FUNCTION_BLOCK "GCS7_E_AnalogInput"	// FB 19
TITLE = Analog Input
//  
//COPYRIGHT:    (C) 2000 BY  BUHLER AG,  CH-9240 UZWILn  SWITZERLAND
//
//PRODUCT:      GCS7
//
//TITLE:        Element Analog Input
//
//-------------------------------------------------------------------------
//
//IDENT:        AUTHOR:             DEPT:                       DATE:
//
//FB19.1.5      A. Egli             CT3                         06-Oct-2008
//              ParMonTimeL=0 or ParMonTimeH=0 are also valide values
//FB19.1.4      A. Egli             CT3                         08-Mar-2005
//              Check ParLimitL > ParLimitLL and ParLimitH < ParLimitHH
//FB19.1.3      A. Egli             CT3                         24-Jan-2005
//              InDisable
//FB19.1.2      A. Egli             CT3                         26-Nov-2001
//              PCDirect Control: Length data is 80 byte not 40 
//FB19.1.1      A. Egli             CT3                         26-Nov-2001
//              Transition StL -->StLL ,StH -->StHH
//FB19.1.0      A. Egli             CT3                         22-Oct-2001
//              New Version of Anlaog Input
//
//-------------------------------------------------------------------------
//
//PURPOSE:      MANUAL : see [AIxxMAN]
//
//RESTRICTIONS: Use the CALL command to call the element
//              e.g. CALL "Element1"
//
//-------------------------------------------------------------------------
//
//MaxDigits:     Siemens: 27'648/ Wago: 32'767
//
//=======================================================
//Log Message: 
//------------------------------------------------------
//1StLLrange LL
//2StLrange L
//3StMidrange Mid
//4StHrange H
//5StHHrange HH
//7fault AI
//8fault device
//9fault cancelled
//11prealarm LL
//12prealarm LL
//13prealarm LL
//14prealarm LL
//15prealarm HH
//21fault LL
//22fault L
//23fault Mid
//24fault H
//25fault HH
//
//=======================================================
//StCode:  State               
//------------------------------------------------------
//  1   StLL                      range LL
//  2   StL                       range L
//  3   StMiddle                  range middle
//  4   StH                       range H
//  5   StHH                      range HH
//
// 11   StLL.Warning              range LL Warning
// 12   StL.Warning               range L  Warning 
// 13   StMiddle                  range middle Warning
// 14   StH.Warning               range H  Warning
// 15   StHH.Warning              range HH Warning
//
// 21   StLL.Faulted              range LL Faulted
// 22   StL.Faulted               range L  Faulted
// 23   StMiddle.Faulted          range middle Faulted
// 24   StH.Faulted               range H  Faulted 
// 25   StHH.Faulted              range HH Faulted
//
// 41   StLL.HWStop               range LL HWStop
// 42   StL.HWStop                range L  HWStop
// 43   StMiddle.HWStop           range middle HWStop
// 44   StH..HWStop               range H  HWStop
// 45   StHH..HWStop              range HH HWStop
//
// 51   StLL.DPFault              range LL DPFault
// 52   StL.DPFault               range L  DPFault
// 53   StMiddle.DPFault          range middle DPFault
// 54   StH..DPFault              range H  DPFault
// 55   StHH..DPFault             range HH DPFault
//
//
// 29   StFaultAI.Dev             fault Device Passiv
// 30   StFaultAI.Input           fault Input  Passiv
// 31   StFaultAI.Dev             fault Device Active
// 32   StFaultAI.Input           fault Input  Active
//
//
//
AUTHOR : EA
FAMILY : GCS7LL
NAME : EL_AI2
VERSION : 1.5
VAR
  StCode : INT ;	//Element state code
  InMonLL : BOOL ;	//After t1 value must be <>StLL, otherwise it is a process fault
  InMonL : BOOL ;	//After t2 value must be <>StL, otherwise it is a process fault
  InMonMid : BOOL ;	//After t3 value must be <>StMid, otherwise it is a process fault
  InMonH : BOOL ;	//After t4 value must be <>StH, otherwise it is a process fault
  InMonHH : BOOL ;	//After t5 value must be <>StHH, otherwise it is a process fault
  spare0205 : BOOL ;
  InpFaultAI : BOOL ;	//Digital input:Fault A/D converter WAGO
  InpFaultDev : BOOL ;	//Digital input Fault device
  InHWStop : BOOL ;	//HW stop is detected, no fault
  InDPFault : BOOL ;	//DP-Fault is detected, no fault
  InDisable : BOOL ;	//Element is disabled
  CmdFaultReset : BOOL ;	//Command to reset fault
  InLocal : BOOL ;	//Local mode
  spare0305 : BOOL ;
  InReport : BOOL ;	//Report all state transitions
  spare0307 : BOOL ;
  OutLL : BOOL ;	//Internal used InValue >= Limit Low Low
  OutL : BOOL ;	//Internal used InValue >= Limit Low
  OutH : BOOL ;	//Internal used InValue >= Limit High
  OutHH : BOOL ;	//Internal used InValue >= Limit High High
  OutOverflow : BOOL ;	//InpValue >32767
  spare0405 : BOOL ;
  OutFaultAI : BOOL ;	//Fault analog input signal
  spare0407 : BOOL ;
  StLL : BOOL ;	//InValue < ParLimitLL (with delay time)
  StL : BOOL ;	//InValue < ParLimitL  (with delay time)
  StMid : BOOL ;	//ParLimitL < InValue < ParLimitH (with delay time)
  StH : BOOL ;	//InValue  > ParLimitH (with delay time)
  StHH : BOOL ;	//InValue  > ParLimitHH (with delay time)
  StFaultAI : BOOL ;	//Fault of analog input value (InpFaultDev or OutFaultAI)
  OutWarning : BOOL ;	//Substate StCode Xxxx.Warning
  OutFaulted : BOOL ;	//Substate StCode Xxxx.Fault
  InpValue : INT ;	//Actual value of analog input
  OutValuePc : INT ;	//Converted InValue in [0.01 %]
  OutValueUnits : DINT ;	//Converted InValue in units
  Msg : STRUCT 	//Read by WinCC
   WarningDoneLL : BOOL ;
   WarningDoneL : BOOL ;
   WarningDoneMid : BOOL ;
   WarningDoneH : BOOL ;
   WarningDoneHH : BOOL ;
   FaultDoneLL : BOOL ;
   FaultDoneL : BOOL ;
   FaultDoneMid : BOOL ;
   FaultDoneH : BOOL ;
   FaultDoneHH : BOOL ;
   FaultDoneDev : BOOL ;
   FaultDoneAI : BOOL ;
  END_STRUCT ;
  OutAlarmNrLog : INT ;	//Last textnumber send to log
  Par : STRUCT
   ParObjectNo : INT ;	//Is used for communication with PC, e.g. for message
   ParMsgType : INT ;	//Is used for message (translation of state)
   ParHornCode : INT ;	//Is used by horn module
   ParLogOff : BOOL ;	//Report is off
   ParSpare0401 : BOOL ;
   ParValueByUser : BOOL ;	//User writes value direct to OutValueUnits
   ParLimitsPc : BOOL ;	//Limits in percent not in units.
   ParWago : BOOL ;	//Format of analog value is WAGO
   ParNoHornByWarning : BOOL ;	//No alarm horn by warning
   ParWarningLL : BOOL ;	//1=Warning / 0=Fault
   ParWarningL : BOOL ;	//1=Warning / 0=Fault
   ParWarningMid : BOOL ;	//1=Warning / 0=Fault
   ParWarningH : BOOL ;	//1=Warning / 0=Fault
   ParWarningHH : BOOL ;	//1=Warning / 0=Fault
   ParPreAlarmLL : BOOL ;	//Immediately Alarm (Horn and report), if value out of monitored range (after t0.
   ParPreAlarmL : BOOL ;	//Immediately Alarm (Horn and report), if value out of monitored range (after t0.
   ParPreAlarmMid : BOOL ;	//Immediately Alarm (Horn and report), if value out of monitored range (after t0.
   ParPreAlarmH : BOOL ;	//Immediately Alarm (Horn and report), if value out of monitored range (after t0.
   ParPreAlarmHH : BOOL ;	//Immediately Alarm (Horn and report), if value out of monitored range (after t0.
   ParUnitsByZeroDigit : DINT ;	//Zero set point of AD-Converter in units
   ParUnitsByMaxDigit : DINT ;	//Max set point of AD-Converter in units
   ParUnitsBy100Pc : DINT ;	//100 Pc set point of precess working range in units
   ParLimitLL : DINT ;	//LL limit value in units or percent
   ParLimitL : DINT ;	//L limit value in units or percent
   ParLimitH : DINT ;	//H limit value in units or percent
   ParLimitHH : DINT ;	//HH limit value in units or percent
   ParMonTimeLL : INT ;	//t1: At end of t1 InValue has to be <> StLL, otherwise StFault.
   ParMonTimeL : INT ;	//t1: At end of t1 InValue has to be <> StL, otherwise StFault.
   ParMonTimeMid : INT ;	//t2: At end of t2 InValue has to be <> StMid, otherwise StFault.
   ParMonTimeH : INT ;	//t2: At end of t2 InValue has to be <> StH, otherwise StFault.
   ParMonTimeHH : INT ;	//t3: At end of t3 InValue has to be <> StHH, otherwise StFault.
   ParDelayTimeDown : INT  := 20;	//Delay time until element changes to the lower state
   ParDelayTimeUp : INT  := 20;	//Delay time until element changes to the higher state
   ParDelayTime : INT ;	//Requested fault delay time (InpFaultAI, InpFaultDev)
   OutMonTimeLL : INT ;	//Actual time: monitoring
   OutMonTimeL : INT ;	//Actual time: monitoring
   OutMonTimeMid : INT ;	//Actual time: monitoring
   OutMonTimeH : INT ;	//Actual time: monitoring
   OutMonTimeHH : INT ;	//Actual time: monitoring
   OutDelayTimeDown : INT ;	//Actual time: delay
   OutDelayTimeUp : INT ;	//Actual time: delay
   OutDelayTime : INT ;	//Actual time: DelayTime
   Spare66 : INT ;
  END_STRUCT ;
END_VAR
VAR_TEMP
  tmpStoreAR2 : DWORD ;	//store the Instance Pointer
  tmpLenDyn : DINT ;
  tmpLOGvalue : WORD ;	//LOG value
  tmpReport : BOOL ;	//Global LOG all
  tmpDConverter : REAL ;	//provisional result: ParUnitsByMaxDigit - ParUnitsByZeroDigit
  tmpDProcess : REAL ;	//provisional result: ParUnitsBy100Pc - ParUnitsByZeroDigit
  tmpLimitMinPc : REAL ;	//Limit minimum in percent
  tmpLimitMaxPc : REAL ;	//Limit maximum in percent
  tmpInpValue : REAL ;	//store actual value
  tmpFaultAI : BOOL ;
  tmpLocal : BOOL ;
  tmpHornOn : BOOL ;
END_VAR
BEGIN
NETWORK
TITLE = Start Global
      L     88;
      T     #tmpLenDyn;	//--> Len dynamic data in byte
//---Report is on---
      O     "GCS7_Gr_OutReportAll";	//---Global OutReportAll
      O     #InReport;
      =     #tmpReport;
//--Local ------------
      A     #InLocal;
      O     #InHWStop;
      O     #InDPFault;
      O     #InDisable;	//[1.3]
      =     #tmpLocal;
//-----------------
      SET;
      R     #tmpHornOn;
NETWORK
TITLE = PC Control
      L     "SYS_DirectCtrlDB".PC.ObjectNo;	//PCControl.ObjectNo
      L     #Par.ParObjectNo;	//Input ObjectNo
      <>I;
      JC    Ctrl;
//=== Test OType      ========================
      L     1019;	//Input object type
      L     "SYS_DirectCtrlDB".PC.ObjectType;	//PCControl.ObjectType
      <>I;
      JC    Ctrl;
//=== Test Handshake =========================
      A     "SYS_DirectCtrlDB".PC.Hsk.FExamine;	//PC.Hsk.FExamine
      JC    pExa;
      A     "SYS_DirectCtrlDB".PC.Hsk.FDefineCmd;	// PC.Hsk.FDefineCmd
      JC    pCmd;
      A     "SYS_DirectCtrlDB".PC.Hsk.FDefinePara;	//PC.Hsk.FDefinePara
      JC    pPar;
pIni: L     2;	// FcInit
      UC    "SYS_DirectCtrl";
      JU    Ctrl;
// Write parameter 
pPar: LAR1  P#DBX 58.0;
      L     P##Par;
      L     DW#16#FFFFF;
      AD;
      +AR1;
      L     DBD [AR1,P#20.0];
      T     #Par.ParLimitLL;
      L     DBD [AR1,P#24.0];
      T     #Par.ParLimitL;
      L     DBD [AR1,P#28.0];
      T     #Par.ParLimitH;
      L     DBD [AR1,P#32.0];
      T     #Par.ParLimitHH;
      L     DBW [AR1,P#36.0];
      T     #Par.ParMonTimeLL;
      L     DBW [AR1,P#38.0];
      T     #Par.ParMonTimeL;
      L     DBW [AR1,P#40.0];
      T     #Par.ParMonTimeMid;
      L     DBW [AR1,P#42.0];
      T     #Par.ParMonTimeH;
      L     DBW [AR1,P#44.0];
      T     #Par.ParMonTimeHH;
      L     DBW [AR1,P#46.0];
      T     #Par.ParDelayTimeDown;
      L     DBW [AR1,P#48.0];
      T     #Par.ParDelayTimeUp;
      L     DBW [AR1,P#50.0];
      T     #Par.ParDelayTime;
// Write new commands from PC to Interface object
pCmd: A     "SYS_DirectCtrlDB".PC.Cmd1[11];	//Cmd1[11]=CmdFaultReset
      S     #CmdFaultReset;
      A     "SYS_DirectCtrlDB".PC.Cmd1[14];	//Cmd1[14]=CmdReportOn
      S     #InReport;
      A     "SYS_DirectCtrlDB".PC.Cmd2[14];	//Cmd2[14]=CmdReportOff
      R     #InReport;
      JU    pIni;
pExa: TAR2;	// Address Dynamic datas
      T     "SYS_DirectCtrlDB".GC.InDynAddr;	// -->PCControl.GC.InDynAddr
      L     #tmpLenDyn;	// Length Dynamic datas
      T     "SYS_DirectCtrlDB".GC.InDynLen;	// -->PCControl.GC.InDynLen
      L     "SYS_DirectCtrlDB".GC.InDynAddr;	// Address Parameters
      T     "SYS_DirectCtrlDB".GC.InParaAddr;	// -->PCControl.GC.InParaAddr
      L     0;	// Length parameter
      T     "SYS_DirectCtrlDB".GC.InParaLen;	// -->PCControl.GC.InParaLen
      L     1;	// Code FcExamine
      UC    "SYS_DirectCtrl";
Ctrl: NOP   0;
NETWORK
TITLE = Global Value Calculation
//                   InpValue    
// OutValueUnits =   -------- * (ParUnitsByMaxDigit- ParUnitsByZeroDigit) 
//+ParUnitsByZeroDigit
//                   maxDigits     
//                     
// OutValuePc    =   (OutValueUnits / ParUnitsBy100Pc) *10'000
//                     
      AN    #Par.ParValueByUser;
      JC    aiJ1;
      L     #OutValueUnits;	// Value by user software
      DTR;
      JU    aiPc;
aiJ1: L     32767;
      L     #InpValue;
      ==I;
      AN    #Par.ParWago;
      =     #OutOverflow;
      L     -32767;
      <=I;
      AN    #Par.ParWago;
      O     #InpFaultAI;
      =     #OutFaultAI;	//--> Wireing broken of underflow analog input
      L     0.000000e+00;
      JC    aiNO;	// aip0
      L     #InpValue;
      ITD;
      DTR;
      A     #Par.ParWago;
      JC    aiJw;
      L     2.764800e+04;	// Max number of digits SIEMENS          
      JU    aiJc;
aiJw: L     3.276700e+04;	// Max number of digits WAGO             
aiJc: /R;
      T     #tmpInpValue;
      L     #Par.ParUnitsByMaxDigit;
      L     #Par.ParUnitsByZeroDigit;
      -D;
      DTR;
      L     #tmpInpValue;
      *R;
      L     #Par.ParUnitsByZeroDigit;
      DTR;
      +R;
      T     #tmpInpValue;
      RND;	// Real to Integer
      T     #OutValueUnits;
      L     #tmpInpValue;
aiPc: L     #Par.ParUnitsBy100Pc;
      DTR;
      /R;
      L     1.000000e+04;
      *R;
      RND;	// Real to Integer
      T     #OutValuePc;
aiNO: NOP   0;
NETWORK
TITLE = Test limits
      L     #OutValuePc;
      ITD;
      A     #Par.ParLimitsPc;
      JC    bLL;
      L     #OutValueUnits;
bLL:  L     #Par.ParLimitLL;
      >=D;
      =     #OutLL;
// 
      L     #OutValuePc;
      ITD;
      A     #Par.ParLimitsPc;
      JC    bL;
      L     #OutValueUnits;
bL:   L     #Par.ParLimitL;
      >=D;
      A     #OutLL;	//[1.4]
      =     #OutL;
// 
      L     #OutValuePc;
      ITD;
      A     #Par.ParLimitsPc;
      JC    bHH;
      L     #OutValueUnits;
bHH:  L     #Par.ParLimitHH;
      >D;
      =     #OutHH;
// 
      L     #OutValuePc;
      ITD;
      A     #Par.ParLimitsPc;
      JC    bH;
      L     #OutValueUnits;
bH:   L     #Par.ParLimitH;
      >D;
      O     #OutHH;	//[1.4]
      =     #OutH;
//---Report is on---
      O     "GCS7_Gr_OutReportAll";	//---Global OutReportAll
      O     #InReport;
      =     #tmpReport;
NETWORK
TITLE = Fault delay time: ParDelayTime 
//Test or Running delay time ====================
//---Condition for Delay Fault
      A     #InpFaultDev;
      O     #OutFaultAI;
      AN    #tmpLocal;
      JC    TFF1;
      R     #tmpFaultAI;
      L     0;
      T     #Par.OutDelayTime;
      JU    TFF0;
TFF1: AN    "GCS7_Gr_OutTick200ms";	// Decrement all 200ms
      L     #Par.OutDelayTime;
      JC    TFF3;
      +     2;
TFF3: T     #Par.OutDelayTime;
      L     #Par.ParDelayTime;
      >=I;
      =     #tmpFaultAI;
      JCN   TFF0;
      T     #Par.OutDelayTime;
TFF0: NOP   0;
NETWORK
TITLE = Count Delay Timer
      AN    "GCS7_Gr_OutTick500ms";	//Gr.OutTick500ms
      JC    DTJ0;
      L     #Par.OutDelayTimeDown;
      +     5;	//Increment all 500ms
      T     #Par.OutDelayTimeDown;
      L     #Par.OutDelayTimeUp;
      +     5;	//Increment all 500ms
      T     #Par.OutDelayTimeUp;
DTJ0: NOP   0;
NETWORK
TITLE = FaultReset
      AN    #CmdFaultReset;	//---Condition for StFault
      AN    "GCS7_Gr_OutFaultReset";	// Gr.OutFaultReset
      AN    #InLocal;
      JC    FREn;
      R     #Msg.WarningDoneLL;
      R     #Msg.WarningDoneL;
      R     #Msg.WarningDoneMid;
      R     #Msg.WarningDoneH;
      R     #Msg.WarningDoneHH;
      R     #Msg.FaultDoneLL;
      R     #Msg.FaultDoneL;
      R     #Msg.FaultDoneMid;
      R     #Msg.FaultDoneH;
      R     #Msg.FaultDoneHH;
      R     #Msg.FaultDoneAI;
      R     #Msg.FaultDoneDev;
//--- Message Fault Cancelled---------------
      A     #Par.ParLogOff;
      ON    #OutFaulted;
      R     #OutFaulted;
      JC    FREn;
      R     #OutFaulted;
      L     B#(3, 9);	// MessageClass Operater "fault cancelled"
      T     #tmpLOGvalue;
      CALL  "GCS7_LogConvert" (
           ObjectNo                 := #Par.ParObjectNo,
           MsgType                  := #Par.ParMsgType,
           ClassMsgTxt              := #tmpLOGvalue,
           OType                    := 1019);	// LOG Message Converter / Entry / Contains Class and TextNo
FREn: NOP   0;
NETWORK
TITLE = Init States
      AN    #StLL;
      AN    #StL;
      AN    #StMid;
      AN    #StH;
      AN    #StHH;
      AN    #StFaultAI;
      JCN   InEn;
///=====================================
//Init after download DB
///=====================================
//Condition for StHH
      A     #OutHH;
      JC    xxHH;
//Condition for StH
      A     #OutH;
      JC    xx_H;
//Condition for StMid
      A     #OutL;
      JC    xxMi;
//Condition for StL
      A     #OutLL;
      JC    xx_L;
//Condition for StLL
      JU    xxLL;
InEn: NOP   0;
NETWORK
TITLE = StLL
      AN    #StLL;
      JC    LLEn;
      JU    LL;
//===============================================
//Transition  to StLL
//===============================================
xxLL: SET;
      S     #StLL;	//Initialise: goto StLL
      L     0;
      T     #Par.OutDelayTimeUp;
      AN    #InReport;
      JC    LLEn;
      L     B#(4, 1);	// Message ('Low Low' )
      JU    Log;
//===============================================
//Logic
//===============================================
//Init
LL:   AN    #InMonLL;
      R     #OutWarning;
      L     0;
      T     #Par.OutDelayTimeDown;
      A     #OutLL;
      JC    LLJ1;
      L     0;
      T     #Par.OutDelayTimeUp;
//---1. Condition for StFault
LLJ1: A     #tmpFaultAI;
      R     #StLL;
      JC    xxFI;
//---Condition for StL
      L     #Par.ParDelayTimeUp;
      L     #Par.OutDelayTimeUp;
      <=I;
      A     #OutLL;	//Change with delay
      O     #OutL;	//Immediate change
      R     #StLL;
      JC    xx_L;
LLEn: NOP   0;
NETWORK
TITLE = Monitoring LL
      AN    #OutLL;
      A     #InMonLL;
      AN    #tmpLocal;
      JC    mLL1;
      L     #Par.ParMonTimeLL;
      T     #Par.OutMonTimeLL;
      JU    mLL0;
mLL1: AN    "GCS7_Gr_OutTick500ms";	//Gr.OutTick500ms
      L     #Par.OutMonTimeLL;
      JC    mLL2;
      L     5;
      -I;	// Decrement all 500ms
      JP    mLL2;
      L     0;
mLL2: T     #Par.OutMonTimeLL;
//----------------------------------------
//FaultLL
//----------------------------------------
      L     #Par.OutMonTimeLL;
      L     0;
      <=I;
      AN    #Par.ParWarningLL;
      JCN   mLLP;
      S     #OutFaulted;
      AN    #Msg.FaultDoneLL;
      S     #Msg.FaultDoneLL;
      S     #tmpHornOn;
      L     B#(1, 21);	// MessageClass Error "fault Low Low"
      JC    Log;
//----------------------------------------
//PreAlarm/WarningLL
//----------------------------------------
mLLP: L     #Par.OutMonTimeLL;
      L     0;
      <=I;
      O     #Par.ParPreAlarmLL;
      JCN   mLL0;
      S     #OutWarning;
      AN    #Msg.FaultDoneLL;
      AN    #Msg.WarningDoneLL;
      JCN   mLL0;
      S     #Msg.WarningDoneLL;
      AN    #Par.ParNoHornByWarning;
      S     #tmpHornOn;
      L     B#(1, 11);	// MessageClass Error "warning Low Low"
      JC    Log;
mLL0: NOP   0;
NETWORK
TITLE = StL
      AN    #StL;
      JC    _LEn;
      JU    _L;
//===============================================
//Transition  to StL
//===============================================
xx_L: SET;
      S     #StL;
      R     #Msg.WarningDoneLL;
      L     0;
      T     #Par.OutDelayTimeDown;
      T     #Par.OutDelayTimeUp;
      AN    #InReport;
      JC    _LEn;
      L     B#(4, 2);	// Message ('Low' )
      JU    Log;
//===============================================
//Logic
//===============================================
//Init
_L:   AN    #InMonL;
      R     #OutWarning;
      AN    #OutLL;
      JC    _LJ1;
      L     0;
      T     #Par.OutDelayTimeDown;
_LJ1: A     #OutL;
      JC    _LJ2;
      L     0;
      T     #Par.OutDelayTimeUp;
//---Condition for StFault
_LJ2: A     #tmpFaultAI;
      R     #StL;
      JC    xxFI;
//---Condition for StLL
      L     #Par.ParDelayTimeDown;
      L     #Par.OutDelayTimeDown;
      <=I;
      AN    #OutLL;	//Change with delay  [1.1]
      R     #StL;
      JC    xxLL;
//---Condition for StMid
      L     #Par.ParDelayTimeUp;
      L     #Par.OutDelayTimeUp;
      <=I;
      A     #OutL;	//Change with delay
      O     #OutH;	//Immediate change
      R     #StL;
      JC    xxMi;
_LEn: NOP   0;
NETWORK
TITLE = Monitoring L
      A(;
      AN    #OutL;
      A     #InMonLL;
      O;
      A     #OutLL;
      AN    #InMonLL;
      );
      A     #InMonL;
      AN    #tmpLocal;
      JC    m_L1;
//==not Monitoring L =================================
      L     #Par.ParMonTimeL;
      T     #Par.OutMonTimeL;
      JU    m_L0;
//==Monitoring L =================================
m_L1: AN    "GCS7_Gr_OutTick500ms";	//Gr.OutTick500ms
      L     #Par.OutMonTimeL;
      JC    m_L2;
      L     5;
      -I;	// Decrement all 500ms
      JP    m_L2;
      L     0;
m_L2: T     #Par.OutMonTimeL;
//----------------------------------------
//FaultL
//----------------------------------------
      L     #Par.OutMonTimeL;
      L     0;
      <=I;
      AN    #Par.ParWarningL;
      AN    #OutL;	//[1.5]
      JCN   m_LP;
      S     #OutFaulted;
      AN    #Msg.FaultDoneLL;
      AN    #Msg.FaultDoneL;
      S     #Msg.FaultDoneL;
      S     #tmpHornOn;
      L     B#(1, 22);	// MessageClass Error "fault Low"
      JC    Log;
//----------------------------------------
//PreAlarm/WarningL
//----------------------------------------
m_LP: L     #Par.OutMonTimeL;
      L     0;
      <=I;
      O     #Par.ParPreAlarmL;
      AN    #OutL;	//[1.5]
      JCN   m_L0;
      S     #OutWarning;
      AN    #Msg.FaultDoneL;
      AN    #Msg.FaultDoneLL;
      AN    #Msg.WarningDoneL;
      AN    #Msg.WarningDoneLL;
      JCN   m_L0;
      S     #Msg.WarningDoneL;
      AN    #Par.ParNoHornByWarning;
      S     #tmpHornOn;
      L     B#(1, 12);	// MessageClass Error "warning Low"
      JC    Log;
m_L0: NOP   0;
NETWORK
TITLE = StMid
      AN    #StMid;
      JC    MiEn;
      JU    Mi;
//===============================================
//Transition  to StMid
//===============================================
xxMi: SET;
      S     #StMid;
      R     #Msg.WarningDoneMid;
      R     #Msg.WarningDoneL;
      R     #Msg.WarningDoneH;
      L     0;
      T     #Par.OutDelayTimeDown;
      T     #Par.OutDelayTimeUp;
      AN    #InReport;
      JC    MiEn;
      L     B#(4, 3);	// Message ('Normal' )
      JU    Log;
//===============================================
//Logic
//===============================================
//Init
Mi:   AN    #InMonMid;
      R     #OutWarning;
      AN    #OutL;
      JC    MiJ1;
      L     0;
      T     #Par.OutDelayTimeDown;
MiJ1: A     #OutH;
      JC    MiJ2;
      L     0;
      T     #Par.OutDelayTimeUp;
//---Condition for StFault
MiJ2: A     #tmpFaultAI;
      R     #StMid;
      JC    xxFI;
//---Condition for StL
      L     #Par.ParDelayTimeDown;
      L     #Par.OutDelayTimeDown;
      <=I;
      AN    #OutL;	//Change with delay
      ON    #OutLL;	//Immediate change
      R     #StMid;
      JC    xx_L;
//---Condition for StH
      L     #Par.ParDelayTimeUp;
      L     #Par.OutDelayTimeUp;
      <=I;
      A     #OutH;	//Change with delay
      O     #OutHH;	//Immediate change
      R     #StMid;
      JC    xx_H;
MiEn: NOP   0;
NETWORK
TITLE = Monitoring Middle
      A(;
      AN    #OutH;
      AN    #InMonHH;
      O;
      A     #OutL;
      A     #InMonHH;
      );
      A     #InMonMid;
      AN    #tmpLocal;
      JC    mMi1;
//==not Monitoring Middle =================================
      L     #Par.ParMonTimeMid;
      T     #Par.OutMonTimeMid;
      JU    mMi0;
//==Monitoring Middle =================================
mMi1: AN    "GCS7_Gr_OutTick500ms";	//Gr.OutTick500ms
      L     #Par.OutMonTimeMid;
      JC    mMi2;
      L     5;
      -I;	// Decrement all 500ms
      JP    mMi2;
      L     0;
mMi2: T     #Par.OutMonTimeMid;
//----------------------------------------
//FaultMid
//----------------------------------------
      L     #Par.OutMonTimeMid;
      L     0;
      <=I;
      AN    #Par.ParWarningMid;
      JCN   mMiP;
      S     #OutFaulted;
      AN    #Msg.FaultDoneMid;
      S     #Msg.FaultDoneMid;
      S     #tmpHornOn;
      L     B#(1, 23);	// MessageClass Error "fault Mid"
      JC    Log;
//----------------------------------------
//PreAlarm / WarningMid
//----------------------------------------
mMiP: L     #Par.OutMonTimeMid;
      L     0;
      <=I;
      O     #Par.ParPreAlarmMid;
      JCN   mMi0;
      S     #OutWarning;
      AN    #OutFaulted;
      AN    #Msg.WarningDoneMid;
      JCN   mMi0;
      S     #Msg.WarningDoneMid;
      AN    #Par.ParNoHornByWarning;
      S     #tmpHornOn;
      L     B#(1, 13);	// MessageClass Error "warning mid"
      JC    Log;
mMi0: NOP   0;
NETWORK
TITLE = StH
      AN    #StH;
      JC    _HEn;
      JU    _H;
//===============================================
//Transition  to StH
//===============================================
xx_H: SET;
      S     #StH;
      R     #Msg.WarningDoneHH;
      L     0;
      T     #Par.OutDelayTimeDown;
      T     #Par.OutDelayTimeUp;
      AN    #InReport;
      JC    _HEn;
      L     B#(4, 4);	// Message ('High' )
      JU    Log;
//===============================================
//Logic
//===============================================
//Init
_H:   AN    #InMonH;
      R     #OutWarning;
      AN    #OutH;
      JC    _HJ1;
      L     0;
      T     #Par.OutDelayTimeDown;
_HJ1: A     #OutHH;
      JC    _HJ2;
      L     0;
      T     #Par.OutDelayTimeUp;
//---Condition for StFault
_HJ2: A     #tmpFaultAI;
      R     #StH;
      JC    xxFI;
//---Condition for StMid
      L     #Par.ParDelayTimeDown;
      L     #Par.OutDelayTimeDown;
      <=I;
      AN    #OutH;	//Change with delay
      ON    #OutL;	//Immediate change
      R     #StH;
      JC    xxMi;
//---Condition for StHH
      L     #Par.ParDelayTimeUp;
      L     #Par.OutDelayTimeUp;
      <=I;
      A     #OutHH;	//Change with delay [1.1]
      R     #StH;
      JC    xxHH;
_HEn: NOP   0;
NETWORK
TITLE = Monitoring H
      A(;
      AN    #OutHH;	//Monitoring < HH
      AN    #InMonHH;
      O;
      A     #OutH;	//Monitoring >H
      A     #InMonHH;
      );
      A     #InMonH;
      AN    #tmpLocal;
      JC    m_H1;
//==not Monitoring H =================================
      L     #Par.ParMonTimeH;
      T     #Par.OutMonTimeH;
      JU    m_H0;
//==Monitoring H =================================
m_H1: AN    "GCS7_Gr_OutTick500ms";	//Gr.OutTick500ms
      L     #Par.OutMonTimeH;
      JC    m_H2;
      L     5;
      -I;	// Decrement all 500ms
      JP    m_H2;
      L     0;
m_H2: T     #Par.OutMonTimeH;
//----------------------------------------
//Fault High 
//----------------------------------------
      L     #Par.OutMonTimeH;
      L     0;
      <=I;
      AN    #Par.ParWarningH;
      A     #OutH;	//Monitoring >H [1.5]
      JCN   m_HP;
      S     #OutFaulted;
      AN    #Msg.FaultDoneHH;
      AN    #Msg.FaultDoneH;
      S     #Msg.FaultDoneH;
      S     #tmpHornOn;
      L     B#(1, 24);	// MessageClass Error "fault high"
      JC    Log;
//----------------------------------------
//PreAlarm  / Warning High
//----------------------------------------
m_HP: L     #Par.OutMonTimeH;
      L     0;
      <=I;
      O     #Par.ParPreAlarmH;
      A     #OutH;	//Monitoring >H [1.5]
      JCN   m_H0;
      S     #OutWarning;
      AN    #Msg.FaultDoneH;
      AN    #Msg.FaultDoneHH;
      AN    #Msg.WarningDoneHH;
      AN    #Msg.WarningDoneH;
      JCN   m_H0;
      S     #Msg.WarningDoneH;
      AN    #Par.ParNoHornByWarning;
      S     #tmpHornOn;
      L     B#(1, 14);	// MessageClass Error "warning high"
      JC    Log;
m_H0: NOP   0;
NETWORK
TITLE = StHH
      AN    #StHH;
      JC    HHEn;
      JU    HH;
//===============================================
//Transition  to StHH
//===============================================
xxHH: SET;
      S     #StHH;
      L     0;
      T     #Par.OutDelayTimeDown;
      AN    #InReport;
      JC    HHEn;
      L     B#(4, 5);	// Message ('High High' )
      JU    Log;
//===============================================
//Logic
//===============================================
//Init
HH:   AN    #InMonHH;
      R     #OutWarning;
      AN    #OutHH;
      JC    HHJ1;
      L     0;
      T     #Par.OutDelayTimeDown;
HHJ1: L     0;
      T     #Par.OutDelayTimeUp;
//---Condition for StFault
      A     #tmpFaultAI;
      R     #StHH;
      JC    xxFI;
//---Condition for StH
      L     #Par.ParDelayTimeDown;
      L     #Par.OutDelayTimeDown;
      <=I;
      AN    #OutHH;	//Change with delay
      ON    #OutH;	//Immediate change
      R     #StHH;
      JC    xx_H;
HHEn: NOP   0;
NETWORK
TITLE = Monitoring HH
      A     #OutHH;
      A     #InMonHH;
      AN    #tmpLocal;
      JC    mHH1;
//==not Monitoring HH =================================
      L     #Par.ParMonTimeHH;
      T     #Par.OutMonTimeHH;
      JU    mHH0;
//==Monitoring HH =================================
mHH1: AN    "GCS7_Gr_OutTick500ms";	//Gr.OutTick500ms
      L     #Par.OutMonTimeHH;
      JC    mHH4;
      L     5;
      -I;	// Decrement all 500ms
      JP    mHH4;
      L     0;
mHH4: T     #Par.OutMonTimeHH;
//----------------------------------------
//Fault High High 
//----------------------------------------
      L     #Par.OutMonTimeHH;
      L     0;
      <=I;
      AN    #Par.ParWarningHH;
      JCN   HHPa;
      S     #OutFaulted;
      AN    #Msg.FaultDoneHH;
      S     #Msg.FaultDoneHH;
      S     #tmpHornOn;
      L     B#(1, 25);	// MessageClass Error "fault high high"
      JC    Log;
//----------------------------------------
//PreAlarm  / Warning High High
//----------------------------------------
HHPa: L     #Par.OutMonTimeHH;
      L     0;
      <=I;
      O     #Par.ParPreAlarmHH;
      JCN   mHH0;
      S     #OutWarning;
      AN    #Msg.FaultDoneHH;
      AN    #Msg.WarningDoneHH;
      JCN   mHH0;
      S     #Msg.WarningDoneHH;
      AN    #Par.ParNoHornByWarning;
      S     #tmpHornOn;
      L     B#(1, 15);	// MessageClass Error "warning high high"
      JC    Log;
mHH0: NOP   0;
NETWORK
TITLE =  StFaultAI
      AN    #StFaultAI;
      JC    FIEn;
      JU    FI;
//===============================================
//Transition  to StHH
//===============================================
xxFI: SET;
      S     #StFaultAI;
      A     #InLocal;
      JC    FIEn;
      S     #OutFaulted;
      S     #tmpHornOn;
      L     B#(1, 8);	// MessageClass Error "fault device"
      A     #InpFaultDev;
      S     #Msg.FaultDoneDev;
      JC    Log;
      L     B#(1, 7);	// MessageClass Error "fault AD"
      S     #Msg.FaultDoneAI;
      JU    Log;
//===============================================
//Logic
//===============================================
//Retry message
FI:   A     #tmpFaultAI;
      AN    #InLocal;
      AN    #OutFaulted;
      JC    xxFI;
//Condition for StFaultAI
      A     #tmpFaultAI;
      JC    FIEn;
      R     #StFaultAI;
//Condition for StHH
      A     #OutHH;
      JC    xxHH;
//Condition for StH
      A     #OutH;
      JC    xx_H;
//Condition for StMid
      A     #OutL;
      JC    xxMi;
//Condition for StL
      A     #OutLL;
      JC    xx_L;
//Condition for StLL
      JU    xxLL;
FIEn: NOP   0;
NETWORK
TITLE = LOG Message
      JU    LoEn;
Log:  A     #Par.ParLogOff;	//---Set LOG Message
      JC    LoEn;
      T     #tmpLOGvalue;
      L     W#16#FF;
      AW;
      T     #OutAlarmNrLog;
      CALL  "GCS7_LogConvert" (
           ObjectNo                 := #Par.ParObjectNo,
           MsgType                  := #Par.ParMsgType,
           ClassMsgTxt              := #tmpLOGvalue,
           OType                    := 1019);	// LOG Message Converter / Entry / Contains Class and TextNo
LoEn: NOP   0;
NETWORK
TITLE = Global End
      CLR;	//---Clear all commands
      =     #CmdFaultReset;
//---Group flag ----------------------------
      A     #OutFaulted;
      R     #OutWarning;
//---Group flag ----------------------------
      A     #InpFaultDev;
      =     #Msg.FaultDoneAI;
      A     #OutFaultAI;
      =     #Msg.FaultDoneAI;
//---Horn On-----------------------------
      AN    #tmpHornOn;
      JC    glJ1;
      S     "GCS7_Gr_InFaultFlag";	// Gr.InFaultFlag
      CALL  "SYS_Horn_Code" (
           FcCode                   := 1,
           ParObjectType            := 1019,
           ParObjectNo              := #Par.ParObjectNo,
           ParHornCode              := #Par.ParHornCode);
glJ1: NOP   0;
//--Output for group 
      A     #InDPFault;
      AN    #InLocal;
      S     "GCS7_Gr_InDPFault";
      A     #InHWStop;
      AN    #InLocal;
      S     "GCS7_Gr_InHWStop";
NETWORK
TITLE = State Code
      A     #InDisable;	//[1.3]
      AN    #OutFaulted;	//[1.3]
      L     6;	// Code: Disabled
      JC    STC;
      L     1;	// Code: range LL
      A     #StLL;
      JC    STC1;
      L     2;	// Code: range L
      A     #StL;
      JC    STC1;
      L     3;	// Code: range middle
      A     #StMid;
      JC    STC1;
      L     4;	// Code: range H
      A     #StH;
      JC    STC1;
      L     5;	// Code: range HH
      A     #StHH;
      JC    STC1;
//--FaultAI.Dev  local
      A     #InLocal;
      A     #InpFaultDev;
      L     29;
      JC    STC;
//--FaultAI.Value local
      A     #InLocal;
      L     30;
      JC    STC;
//--FaultAI.Dev  Active
      A     #InpFaultDev;
      L     31;
      JC    STC;
//--FaultAI.Value Active
      L     32;
      JU    STC;
//Add +20 if Faulted
STC1: AN    #OutFaulted;
      JC    STCH;
      +     20;
      JC    STC;
//Add +40 if HWStop
STCH: AN    #InHWStop;
      JC    STCD;
      +     40;
      JC    STC;
//Add +50 if DPFault
STCD: AN    #InDPFault;
      JC    STCW;
      +     50;
      JC    STC;
//Add +10 if warning
STCW: AN    #OutWarning;
      JC    STC;
      +     10;
STC:  L     #StCode;	// Old state code
      TAK;
      T     #StCode;	// Save state code
      <>I;
      L     3;	// Load code for CBit methode
      CC    "SYS_CBitCtrl";
END_FUNCTION_BLOCK

FUNCTION_BLOCK "GCS7_E_ValveControl4Pos"	// FB 20
TITLE = VLS4
//  
//COPYRIGHT:    (C) 1996 BY  BUHLER LTD.
//                           CH-9240 UZWIL  SWITZERLAND
//
//PRODUCT:      GCS7
//
//TITLE:        ELEMENT Valve control with 3 or 4 position
//              (GCPROVB Revision 13)
//-------------------------------------------------------------------------
//
//IDENT:        AUTHOR:             DEPT:                       DATE:
//
//FB20.7.2      A. Egli             CT3                         19-Mai-2009
//              StCtoHN-->StLN: Reset  Par.tmpOutpHN ,  OutpHold
//FB20.7.1      A. Egli             CT3                         06-Mar-2008
//              PCD: ParTimeControl check Hsk.FDefineValue
//FB20.7.0      A. Egli             CT3                         21-Sep-2007
//              Linak
//FB20.6.2      A. Egli             CT3                         14-Mai-2007
//              ParTimeControl: Do not Set CmdLNMan if CmdHN=1 
//FB20.6.1      A. Egli             CT3                         08-Jun-2006
//              ParTimeControl: PCD
//FB20.6.0      A. Egli             CT3                         15-May-2006
//              ParTimeControl: Measuring middle position be time
//FB20.5.3      A. Egli             CT3                         12-Dec-2005
//              Reset OutWarning also with GCS7_Gr_OutFaultReset 
//FB20.5.2      A. Egli             CT3                         09-Mar-2005
//              Transition StCToLN ot StNoPosition when OutpLN=0
//FB20.5.1      A. Egli             CT3                         13-Oct-2004
//              Transition StNoPosition to StCToLN when InLN=1
//FB20.5.0      A. Egli             CT3                         05-Aug-2004
//              - ParAngle:
//                 1=Positioning from both side 
//                 0=Positioning always from lower number 
//FB20.4.2      A. Egli             CT3                         18-Nov-2003
//              - Alarm-Number for LOG :1,2,3 changed 
//FB20.4.1      A. Egli             CT3                         22-Sep-2003
//              - Check if only one LS pressed 
//FB20.4.0      A. Egli             CT3                         17-Jun-2002
//              - New Release with one block 
//              - StWarning
//FB20.3.0      A. Egli             CT3                         13-Mar-2002
//              ParDFZK : Flap box DFZK-2
//FB20.2.1      A. Egli             CT3                         22-Aug-2000
//              Gr.OutFaultReset
//FB20.2A       A. Egli             CT3                         04-Mai-1998
//              StFault = StCode 32
//FB20.1A       A.Egli              AEE61                       17-Jul-1997
//              1st Release in S7
//
//-------------------------------------------------------------------------
//
//PURPOSE:      MANUAL : see [VLS4xMAN]
//
//RESTRICTIONS: S7
//              ACCU2: Pointer to dynamic datas of the element
//              ACCU1: Pointer to parameter datas of the element
//
//-------------------------------------------------------------------------
//=======================================================
//Log Message: 
//------------------------------------------------------
//O   set position LN
//2   set position HN
//3   set position Middle 1
//4   set position Middle 2
//5   set no position
//9   fault cancelled
//11  fault LN
//12  fault Middle 1 
//13  fault Middle 2
//14  fault HN
//15  fault AI
//
//=======================================================
//StCode:  State               
//------------------------------------------------------
//32   StFault                
// 1   StLN                   
// 2   StCtoHN                
// 3   StHN                    
// 4   StCtoLN                
// 5   StNoPosition                   no position
// 6   StMiddle1              
// 7   StMiddle2              
//11   StLN.StWarning                   
//12   StCtoHN.StWarning                
//13   StHN.StWarning                    
//14   StCtoLN.StWarning                
//15   StNoPosition.StWarning         no position
//16   StMiddle1.StWarning              
//17   StMiddle2.StWarning              
//45   StNoPosition.HWStop            StNoPosition + InHWStop
//55   StNoPosition.DPFault           StNoPosition + InDPFault
//
//
//
//
//
AUTHOR : EA
FAMILY : GCS7LL
NAME : VLS4
VERSION : 7.2
VAR
  StCode : INT ;	//Element state code
  InLN : BOOL ;	//Position LN is requested (1=Set position LN/0=Change to higher position allowed
  CmdMiddle1 : BOOL ;	//Pulse to set position Middle 1 (automatic)
  CmdMiddle2 : BOOL ;	//Pulse to set position Middle 2 (automatic)
  CmdHN : BOOL ;	//Pulse to set position HN       (automatic)
  InpLN : BOOL ;	//Digital input position LN
  InpMiddle1 : BOOL ;	//Digital input position Middle1
  InpMiddle2 : BOOL ;	//Digital input position Middle2
  InpHN : BOOL ;	//Digital input position HN
  CmdLNMan : BOOL ;	//Pulse to move to posotion LN in manual mode
  CmdPrevPos : BOOL ;	//Pulse move to next lower  position in manual mode
  CmdNextPos : BOOL ;	//Pulse move to next higher position in manual mode
  CmdFaultReset : BOOL ;	//Command to reset fault
  InLocal : BOOL ;	//1= Local mode (no fault by start with service switch)
  InManual : BOOL ;	//1= Manual/ 0= Automatic
  InReport : BOOL ;	//Report of all state transitions
  InpFaultAI : BOOL ;	//*AI: Fault Analog Value (Siemens Internal Used)
  InHWStop : BOOL ;	//HW stop is detected, no fault
  InDPFault : BOOL ;	//DP-Fault is detected, no fault
  OutWarning : BOOL ;	//More than 4 re-adjust loop during warning time
  OutpLN2 : BOOL ;	//Digital output (only used for DFZK2)
  OutpHN2 : BOOL ;	//Digital output (only used for DFZK2)
  OutpHold : BOOL ;	//Digital output HOLD, Is TRUE during change to HN or in position Middle1,Middle2
  OutpLN : BOOL ;	//Digital output Valve LN
  OutpHN : BOOL ;	//Digital output Valve HN
  StLN : BOOL ;	//Element is in position LN
  StCtoHN : BOOL ;	//Element is moving to higher position
  StHN : BOOL ;	//Element is in position HN
  StCtoLN : BOOL ;	//Element is moving to lower position
  StFault : BOOL ;	//Element has a fault
  StNoPosition : BOOL ;	//Element is not in a final position
  StMiddle1 : BOOL ;	//Element is in position Middle1
  StMiddle2 : BOOL ;	//Element is in position Middle2
  InpPosition : INT ;	//*AI/*TC/*LK: Analog Input Position [digit]/[0.1s]/[pulse]
  InPositionMiddle : INT ;	//*AI/*TC/*LK: Target Position Middle [0.1%]
  OutPosition : INT ;	//*AI/*TC/*LK: Actual Position [0.1%]
  InpPulse : BOOL ;	//*LK: Edge of pulse signal
  spare12 : INT ;
  OutAlarmNrLog : INT ;	//Last textnumber send to log
  Par : STRUCT
   ParObjectNo : INT ;	//Is used for communication with PC, e.g. for message
   ParMsgType : INT ;	//Is used for message (translation of state)
   ParHornCode : INT ;	//Is used by horn module
   ParLogOff : BOOL ;	//Report is off
   ParManual : BOOL ;	//Manual mode without interlocking
   ParNoLSLN : BOOL ;	//No limit switch LN
   ParNoLSMiddle2 : BOOL ;	//No position Middle2
   ParContinuousHN : BOOL ;	//Continuous signal for output OutpHN in position HN
   ParNoReAdjust : BOOL ;	//Change to StFault by losing final position
   ParDFZK : BOOL ;	//Flap box DFZK
   ParAnalog : BOOL ;	//*AI: 1=Analog ; 0=Digital
   ParWago : BOOL ;	//*AI: 1=Wago   ; 0=Siemens
   ParAngle : BOOL ;	//1=Positioning from both side
   ParTimeControl : BOOL ;	//*TC: 1=Position calcualted by time
   ParLinak : BOOL ;	//*LK: 1=Linak with pulse signal
   ParNoLSHN : BOOL ;	//*LK: 1=No limit switch HN
   ParTransTime : INT ;	//Maximum time to move to final position [0.1 s]
   ParWarningTime : INT ;	//In this time are 4 re-adjust loops allowed [0.1 s]
   ParPulseLN : INT ;	//Switch off delay time if arrive pos LN [0.1 s]
   ParPulseMiddle : INT ;	//Switch off delay time if arrive pos middle1 or middle2 [0.1 s]
   ParPulseHN : INT ;	//Switch off delay time if arrive pos HN   [0.1 s]
   ParUnitsByMaxDigit : INT  := 1000;	//*AI: Max set point of AD-Converter in units  [0.1%]
   ParUnitsByZeroDigit : INT ;	//*AI: Zero set point of AD-Converter in units  [0.1%]
   ParPositionTolerance : INT  := 10;	//*AI/*TC: Tolerace actual position [0.1%]
   ParPositionOpen : INT  := 1000;	//*AI/*TC/*LK: Position Open [0.1%] / [0.1s] / [Pulse]
   ParPositionClosed : INT  := 5;	//*AI: Position Cosed [0.1%]
   spare28 : INT ;
   OutDelayTime : INT ;	//Actual time CtoHN, CtoLN, pulse  [0.1 s]
   OutPosTarget : INT ;	//Target position:0=LN;1=Middle1;2=Middle2;3=HN
   OutCntReAdjust : INT ;	//Number og re-adjust loops
   OutWarningTime : INT ;	//Actual warning time  [0.1 s]
   tmpInPosition : INT ;	//Internal used Copy of InPositionMiddle
   tmpOutpLN : BOOL ;	//Internal used
   tmpOutpHN : BOOL ;	//Internal used
   OutReAdjust : BOOL ;	//Re-adjust loop is active
   OutPulseIsOn : BOOL ;	//Delay time is running, slide in position
  END_STRUCT ;
END_VAR
VAR_TEMP
  tmpLOGvalue : WORD ;	//LOG value
  tmpReport : BOOL ;	//Global LOG all
  tmpLenDyn : DINT ;
  tmpLN : BOOL ;	//Condition for LN
  tmpNext : BOOL ;
  tmpTimeEnd : BOOL ;
  tmpPosValid : BOOL ;
  tmpPosActual : INT ;	//Actual position
  tmpLocal : BOOL ;
  tmpNotInLN : BOOL ;
  tmpCntReAdjustUp : BOOL ;
  tmpMid : BOOL ;
  tmpStateNr : INT ;	//StateNr of actual state
  tmpTargetPosition : INT ;	//Temporare
  tmpLocalFault : BOOL ;
  tmpInpValue : REAL ;
  tmpNoLSMiddle2 : BOOL ;
  tmpInpLN : BOOL ;
  tmpAnalog : BOOL ;
  tmpInpHN : BOOL ;
END_VAR
BEGIN
NETWORK
TITLE =  Start Global
      L     60;
      T     #tmpLenDyn;	//--> Len dynamic data in byte
NETWORK
TITLE = PC Control
//=== Test Object number =====================
      L     "SYS_DirectCtrlDB".PC.ObjectNo;	//PCControl.ObjectNo
      L     #Par.ParObjectNo;	//Input ObjectNo
      <>I;
      JC    Ctrl;
//=== Test OType      ========================
      L     1020;	//Input object type
      L     "SYS_DirectCtrlDB".PC.ObjectType;	//PCControl.ObjectType
      <>I;
      JC    Ctrl;
//=== Test Handshake =========================
      A     "SYS_DirectCtrlDB".PC.Hsk.FExamine;	// Handshake.FExamine
      JC    pExa;
      A     "SYS_DirectCtrlDB".PC.Hsk.FDefineCmd;	// Handshake.FDefineCmd
      O     "SYS_DirectCtrlDB".PC.Hsk.FDefineValue;	// Handshake.FDefineValue [7.3]
      JC    pCmd;
      A     "SYS_DirectCtrlDB".PC.Hsk.FDefinePara;	// Handshake.FDefinePara
      JC    pPar;
pIni: L     2;	// FcInit
      UC    "SYS_DirectCtrl";
      JU    Ctrl;
// Write parameter 
pPar: LAR1  P#DBX 58.0;	//PCControl.Value[1]
      L     P##Par;
      L     DW#16#FFFFF;
      AD;
      +AR1;
      L     DBW [AR1,P#8.0];
      T     #Par.ParTransTime;
      L     DBW [AR1,P#10.0];
      T     #Par.ParWarningTime;
      L     DBW [AR1,P#12.0];
      T     #Par.ParPulseLN;
      L     DBW [AR1,P#14.0];
      T     #Par.ParPulseMiddle;
      L     DBW [AR1,P#16.0];
      T     #Par.ParPulseHN;
// Write new commands from PC to Interface of group 
pCmd: A     "SYS_DirectCtrlDB".PC.Cmd1[8];	//Cmd1[8]   =CmdLNMan
      S     #CmdLNMan;
      A     "SYS_DirectCtrlDB".PC.Cmd1[9];	//Cmd1[1]   =CmdPrevPos
      S     #CmdPrevPos;
      A     "SYS_DirectCtrlDB".PC.Cmd1[10];	//Cmd1[2]   =CmdNextPos
      S     #CmdNextPos;
      A     "SYS_DirectCtrlDB".PC.Cmd1[12];	//Cmd1[2]   =CmdHN
      S     #CmdHN;
      AN    "SYS_DirectCtrlDB".PC.Cmd1[4];	//Cmd1[4]   =CmdCalibrate //[6.0]
      ON    #InManual;	//[6.0]
      ON    #InpHN;	//[6.0]
      O     "GCS7_Gr_OutManualOff";	//Global.OutManualOff    //[6.0]
      JC    pCal;	//[6.0]
      L     #InpPosition;	//[6.0]
      T     #Par.ParPositionOpen;	//[6.0]
pCal: A     "SYS_DirectCtrlDB".PC.Cmd1[11];	//Cmd1[11] =CmdFaultReset
      S     #CmdFaultReset;
      A     "SYS_DirectCtrlDB".PC.Cmd1[13];	//Cmd1[13] =CmdManualOn
      S     #InManual;
      A     "SYS_DirectCtrlDB".PC.Cmd2[13];	//Cmd2[13] =CmdManualOff
      R     #InManual;
      A     "SYS_DirectCtrlDB".PC.Cmd1[14];	//Cmd1[14]=CmdReportOn
      S     #InReport;
      A     "SYS_DirectCtrlDB".PC.Cmd2[14];	//Cmd2[14]=CmdReportOff
      R     #InReport;
      AN    #Par.ParAnalog;	//[6.0]
      AN    #Par.ParTimeControl;	//[6.0]
      AN    #Par.ParLinak;	//[7.0]
      JC    pIni;	//[6.0]
      A     #CmdNextPos;	//[6.0]
      A     #StMiddle1;	//[6.0]
      R     #CmdNextPos;	//[6.0]
      A     #CmdNextPos;	//[6.0]
      A     #StHN;	//[6.0]
      R     #CmdNextPos;	//[6.0]
      S     #CmdPrevPos;	//[6.0]
      A     "GCS7_Gr_OutManualOff";	//Global.OutManualOff
      ON    "SYS_DirectCtrlDB".PC.Hsk.FDefineValue;	//[7.1] PC.Hsk.FDefineValue
      JC    pIni;
      L     0;
      L     "SYS_DirectCtrlDB".PC.Cmd3;	// "SYS_PCControl".PC.Cmd3
      ==I;
      AN    #Par.ParTimeControl;	//[6.1]
      AN    #Par.ParLinak;	//[7.0]
      JC    pIni;
      T     #InPositionMiddle;
      AN    #Par.ParTimeControl;	//[6.1]
      AN    #Par.ParLinak;	//[7.0]
      JC    pIni;	//[6.1]
      L     1000;	//[6.1]
      L     #InPositionMiddle;	//[6.1]
      <=I;	//[6.1]
      S     #CmdHN;	//[6.1]
      L     0;	//[6.1]
      L     #InPositionMiddle;	//[6.1]
      >=I;	//[6.1]
      AN    "SYS_DirectCtrlDB".PC.Cmd1[12];	//Cmd1[2]   =CmdHN     //[6.2]
      AN    "SYS_DirectCtrlDB".PC.Cmd1[4];	//Cmd1[4]   =CmdCalibrate //[6.2]
      S     #CmdLNMan;	//[6.1]
      AN    #CmdHN;	//[6.1]
      AN    #CmdLNMan;	//[6.1]
      AN    "SYS_DirectCtrlDB".PC.Cmd1[4];	//Cmd1[4]   =CmdCalibrate //[6.2]
      S     #CmdMiddle1;	//[6.1]
      JU    pIni;
pExa: TAR2;	// Address Dynamic datas
      T     "SYS_DirectCtrlDB".GC.InDynAddr;	// -->PCControl.GC.InDynAddr
      L     #tmpLenDyn;	// Length Dynamic datas
      T     "SYS_DirectCtrlDB".GC.InDynLen;	// -->PCControl.GC.InDynLen
      L     0;
      T     "SYS_DirectCtrlDB".GC.InParaAddr;	// -->PCControl.GC.InParaAddr
      T     "SYS_DirectCtrlDB".GC.InParaLen;	// -->PCControl.GC.InParaLen
      L     1;	// Code FcExamine
      UC    "SYS_DirectCtrl";
      L     13;	//Revision
      T     "SYS_DirectCtrlDB".GC.Revision;
Ctrl: NOP   0;
NETWORK
TITLE = Convert Position Linak [7.0]
      AN    #Par.ParLinak;	//[7.0]
      JC    lkNO;	//[7.0]
      L     #InpPosition;
      L     0;
      >=I;
      AN    #InpLN;
      JC    lkJ1;
      T     #InpPosition;
lkJ1: L     #InpPosition;
      ITD;
      DTR;
      L     #Par.ParPositionOpen;
      DTR;
      /R;
      L     1.000000e+03;
      *R;
      RND;	// Real to Integer
      T     #OutPosition;
      L     #Par.ParPositionTolerance;
      L     #InPositionMiddle;
      +I;
      L     #OutPosition;
      >=I;
      A(;
      L     #InPositionMiddle;
      >=I;
      );
      AN    #InpLN;
      AN    #InpHN;
      =     #InpMiddle1;
//----------------
      A     #CmdMiddle2;
      R     #CmdMiddle2;
      S     #CmdMiddle1;
lkNO: NOP   0;
NETWORK
TITLE = Convert Position Analog
      AN    #Par.ParAnalog;
      JC    aiNO;
      L     #InpPosition;
      L     -32767;
      <=I;
      AN    #Par.ParWago;
      O;
      A     #Par.ParWago;
      A     #InpFaultAI;
      =     #InpFaultAI;	//--> Wireing broken of underflow analog input
      L     0.000000e+00;
      JC    aiNO;	// aip0
      L     #InpPosition;
      ITD;
      DTR;
      A     #Par.ParWago;
      JC    aiJw;
      L     2.764800e+04;	// Max number of digits SIEMENS          
      JU    aiJc;
aiJw: L     3.276700e+04;	// Max number of digits WAGO             
aiJc: /R;
      T     #tmpInpValue;
      L     #Par.ParUnitsByMaxDigit;
      L     #Par.ParUnitsByZeroDigit;
      -D;
      DTR;
      L     #tmpInpValue;
      *R;
      L     #Par.ParUnitsByZeroDigit;
      DTR;
      +R;
      T     #tmpInpValue;
      RND;	// Real to Integer
      T     #OutPosition;
      L     #OutPosition;
      L     #Par.ParPositionTolerance;
      <I;
      =     #InpLN;
      L     #OutPosition;
      L     #Par.ParPositionOpen;
      >=I;
      =     #InpHN;
      L     #Par.ParPositionTolerance;
      L     #InPositionMiddle;
      +I;
      L     #OutPosition;
      >=I;
      A(;
      L     #InPositionMiddle;
      >=I;
      );
      AN    #InpLN;
      AN    #InpHN;
      =     #InpMiddle1;
//----------------
      A     #CmdMiddle2;
      R     #CmdMiddle2;
      S     #CmdMiddle1;
aiNO: NOP   0;
NETWORK
TITLE = Convert Position Time Control [6.0]
      AN    #Par.ParTimeControl;
      JC    tcNO;
      AN    #InpHN;	//[6.1]
      O     #InManual;	//[6.1]
      JC    tcMX;	//[6.1]
      L     #Par.ParPositionOpen;	//[6.1]
      T     #InpPosition;	//[6.1]
      JU    tcHN;	//[6.1]
tcMX: AN    #OutpHN;
      ON    "GCS7_Gr_OutTick200ms";
      O     #InpHN;
      JC    tcHN;
      L     #InpPosition;
      +     2;
      T     #InpPosition;
//--------------
tcHN: AN    #OutpLN;
      ON    "GCS7_Gr_OutTick200ms";
      JC    tcLN;
      L     #InpPosition;
      +     -2;
      T     #InpPosition;
      NOP   0;
//--------------
tcLN: L     #InpPosition;
      L     0;
      >=I;
      AN    #InpLN;
      JC    tcIn;
      T     #InpPosition;
//--------------
tcIn: L     #InpPosition;
      ITD;
      DTR;
      L     #Par.ParPositionOpen;
      DTR;
      /R;
      L     1.000000e+03;
      *R;
      T     #tmpInpValue;
      RND;	// Real to Integer
      T     #OutPosition;
      L     #Par.ParPositionTolerance;
      L     #InPositionMiddle;
      +I;
      L     #OutPosition;
      >=I;
      A(;
      L     #InPositionMiddle;
      >=I;
      );
      AN    #InpLN;
      AN    #InpHN;
      =     #InpMiddle1;
//----------------
      A     #CmdMiddle2;
      R     #CmdMiddle2;
      S     #CmdMiddle1;
tcNO: NOP   0;
NETWORK
TITLE =  All State Init
//===Clear tmp Variable
//===Global Group Orders===
      A     #Par.ParAnalog;	//[6.0]
      O     #Par.ParTimeControl;	//[6.0]
      O     #Par.ParLinak;	//[7.0]
      =     #tmpAnalog;	//[6.0]
      A     "GCS7_Gr_OutManualOn";	//Gr.OutManualOn
      S     #InManual;
      A     "GCS7_Gr_OutManualOff";	//Gr.OutManualOff
      R     #InManual;
      A     #InManual;
      S     "GCS7_Gr_InManual";	//Gr.InManualMode
      A     #InLocal;
      AN    #InManual;
      =     #tmpLocalFault;
      A     #tmpLocalFault;
      O     #InHWStop;
      O     #InDPFault;
      =     #tmpLocal;
//No LS Middle2
      A     #Par.ParNoLSMiddle2;
      O     #tmpAnalog;	//[6.0]
      =     #tmpNoLSMiddle2;
//---InpHN---
      L     #InpPosition;	//[7.0]
      L     #Par.ParPositionOpen;	//[7.0]
      >=I;	//[7.0]
      A     #Par.ParNoLSHN;	//[7.0]
      A     #Par.ParLinak;	//[7.0]
      O     #InpHN;	//[7.0]
      =     #tmpInpHN;
//---InpLN---
      A     #InpLN;
      AN    #InpMiddle1;	//[4.1]
      AN    #InpMiddle2;	//[4.1]
      AN    #tmpInpHN;	//[4.1][7.0]
      =     #tmpInpLN;	//[4.1]
//---Report is on---
      A     "GCS7_Gr_OutReportAll";	//Gr.OutReportAll
      O     #InReport;
      =     #tmpReport;
//---Enable---
      A     #InLN;
      O     #InLocal;
      AN    #InManual;
      O(;
      A     #InLN;
      AN    #Par.ParManual;
      A     #InManual;
      );
      O     #CmdLNMan;
      =     #tmpLN;
//---Next---
//---automatic StCtoHN
      A     #CmdMiddle1;
      O     #CmdMiddle2;
      O     #CmdHN;
      AN    #tmpLocal;	//[5.0]
      =     #tmpNext;
      A     #tmpCntReAdjustUp;
      R     #tmpCntReAdjustUp;
//--- Calculate OutPosTarget 
//  --Target position manual  
      AN    #InManual;
      JC    AUTO;
      A     #StMiddle1;
      A     #CmdPrevPos;
      O     #StNoPosition;
      O     #tmpLN;
      L     0;	// Target Position = LN
      JC    Ipos;
      A     #StMiddle2;
      A     #CmdPrevPos;
      O;
      A     #StHN;
      A     #tmpNoLSMiddle2;
      A     #CmdPrevPos;
      O;
      A     #CmdNextPos;
      A     #StLN;
      O;
      A     #Par.ParTimeControl;	//[6.1]
      A     #CmdMiddle1;	//[6.1]
      AN    #CmdHN;	//[6.1]
      L     1;	// Target Position = Middle1
      JC    Ipos;
      A     #StHN;
      AN    #tmpNoLSMiddle2;
      A     #CmdPrevPos;
      O;
      A     #StMiddle1;
      AN    #tmpNoLSMiddle2;
      A     #CmdNextPos;
      L     2;	// Target Position = Middle2
      JC    Ipos;
      A     #StMiddle1;
      O     #StMiddle2;
      A     #CmdNextPos;
      O     #CmdHN;	//[6.0]
      L     3;	// Target Position = HN
      JC    Ipos;
      JU    I3;
//  --Target position automatic  
AUTO: A     #tmpLN;
      L     0;	// Target Position = LN
      JC    Ipos;
      A     #CmdMiddle1;
      L     1;	// Target Position = Middle1
      JC    Ipos;
      A     #CmdMiddle2;
      L     2;	// Target Position = Middle2
      JC    Ipos;
      A     #CmdHN;
      L     3;	// Target Position = HN
      JC    Ipos;
      JU    I3;
Ipos: T     #Par.OutPosTarget;
//--- Test actual position 
I3:   AN    #tmpPosValid;
      S     #tmpPosValid;
      A     #InpLN;
      AN    #InpMiddle1;
      AN    #InpMiddle2;
      AN    #tmpInpHN;	//[7.0]
      L     0;	// Actual position = LN
      JC    I4;
      AN    #InpLN;
      A     #InpMiddle1;
      AN    #InpMiddle2;
      AN    #tmpInpHN;	//[7.0]
      L     1;	// Actual position = Middle1
      JC    I4;
      AN    #InpLN;
      AN    #InpMiddle1;
      A     #InpMiddle2;
      AN    #tmpInpHN;	//[7.0]
      L     2;	// Actual position = Middle2
      JC    I4;
      AN    #InpLN;
      AN    #InpMiddle1;
      AN    #InpMiddle2;
      A     #tmpInpHN;	//[7.0]
      L     3;	// Actual position = HN
      JC    I4;
      R     #tmpPosValid;
      L     0;	// Actual position = LN
I4:   T     #tmpPosActual;
//--- Traget Position local mode  
      AN    #tmpLocal;
      JC    INJ1;
      L     #tmpPosActual;
      T     #Par.OutPosTarget;
INJ1: NOP   0;
NETWORK
TITLE = States
//===State machine===
      A     #StLN;
      JC    S0;
      A     #StCtoHN;
      JC    S1;
      A     #StHN;
      JC    S2;
      A     #StCtoLN;
      JC    S3;
      A     #StFault;
      JC    S4;
      A     #StNoPosition;
      JC    S5;
      A     #StMiddle1;
      JC    S6;
      A     #StMiddle2;
      JC    S7;
      S     #StLN;	// Init
      JU    S0;
NETWORK
TITLE = StLN
// Any transition to StLN
xxS0: S     #StLN;
      S     #Par.OutPulseIsOn;
      R     #OutpHold;	//[7.2]
      R     #Par.tmpOutpHN;	//[7.2]
      L     0;
      T     #Par.OutDelayTime;
      AN    #tmpReport;
      JC    OUT;
      L     B#(4, 0);	//MessageClass Info "SET_Closed"
      JU    LOG;
//=== Logic ====
S0:   R     #Par.OutReAdjust;
      AN    #Par.OutPulseIsOn;
      JC    SOJ1;
      AN    "GCS7_Gr_OutTick200ms";	//Gr.OutTick200ms
      L     #Par.OutDelayTime;
      JC    S0T1;
      +     2;
      T     #Par.OutDelayTime;
S0T1: L     #Par.ParPulseLN;
      >=I;
      =     #tmpTimeEnd;
      R     #Par.OutPulseIsOn;
      R     #Par.tmpOutpLN;
// Transition to StCtoHN
SOJ1: A     #tmpNext;
      AN    #InManual;
      AN    #InLocal;
      O;
      A     #InManual;
      A     #CmdLNMan;
      O;
      A     #InManual;
      A     #CmdNextPos;
      O;
      A     #InManual;	//[6.0]
      A     #CmdHN;	//[6.0]
      O;	//[6.1]
      A     #InManual;	//[6.1]
      A     #CmdMiddle1;	//[6.1]
      A     #Par.ParTimeControl;	//[6.1]
      L     #Par.OutPosTarget;
      JC    S0J2;
      L     0;
S0J2: T     #tmpTargetPosition;
      L     0;	//Position LN
      <>I;
      R     #StLN;
      JC    xxS1;	//--> StCtoHN
      <>I;
      A     #tmpPosValid;
      O;
      AN    #Par.ParNoLSLN;
      AN    #tmpInpLN;	//[4.1]
      =     #tmpNotInLN;
// Transition to StCtoLN
      A     #tmpNotInLN;
      AN    #Par.ParNoReAdjust;
      AN    #tmpLocal;
      S     #Par.OutReAdjust;
      S     #tmpCntReAdjustUp;
      R     #StLN;
      JC    xxS3;	//--> StCtoLN
// Transition to StFault
      A     #tmpNotInLN;
      AN    #tmpLocal;
      R     #StLN;
      JC    xxS4;	//--> StFault
// Transition to StNoPos
      A     #tmpNotInLN;
      R     #StLN;
      JC    xxS5;	//--> StNoPosition
      JU    OUT;
NETWORK
TITLE = StCtoHN
// Any transition to StCtoHN
xxS1: S     #StCtoHN;
      R     #Par.tmpOutpLN;
      S     #OutpHold;
      S     #Par.tmpOutpHN;
      AN    #Par.OutPulseIsOn;
      JC    OUT;
      L     0;
      T     #Par.OutDelayTime;
      JU    OUT;
//=== Logic ====
S1:   AN    "GCS7_Gr_OutTick200ms";	//Gr.OutTick200ms
      L     #Par.OutDelayTime;
      JC    S11T;
      +     2;
      T     #Par.OutDelayTime;
S11T: L     #Par.ParTransTime;
      >=I;
      =     #tmpTimeEnd;
      L     #Par.OutPosTarget;
      L     #tmpPosActual;
      ==I;
      A     #tmpPosValid;
      JC    S1J1;
// Transition to StCtoLN;
      L     #Par.OutPosTarget;
      L     #tmpPosActual;
      <I;
      A     #tmpPosValid;
      O;
      A     #tmpTimeEnd;
      AN    #Par.OutReAdjust;
      O(;
      L     #Par.OutPosTarget;
      L     0;	//= StLN
      ==I;
      );
      O(;	//[4.0]
      L     #OutPosition;	//[4.0]
      L     #Par.ParPositionTolerance;	//[4.0]
      -I;	//[4.0]
      L     #InPositionMiddle;	//[4.0]
      >I;	//[4.0]
      A(;
      L     1;	// Target position =StMiddle1
      L     #Par.OutPosTarget;
      ==I;
      );
      A     #tmpAnalog;	//[6.0]//[4.0]
      );	//[4.0]
      S     #Par.OutReAdjust;
      R     #StCtoHN;
      JC    xxS3;	//--> StCtoLN
// Transition to Fault
      A     #tmpTimeEnd;
      R     #StCtoHN;
      JC    xxS4;	//--> StFault
      JU    OUT;
//==Do any Transition   
// Transition to StMiddle1
S1J1: L     1;	// Position StMiddle1
      L     #Par.OutPosTarget;
      ==I;
      R     #StCtoHN;
      JC    xxS6;	//--> StMiddle1
// Transition to StMiddle2
      L     2;	// Position StMiddle2
      L     #Par.OutPosTarget;
      ==I;
      R     #StCtoHN;
      JC    xxS7;	//--> StMiddle2
// Transition to StHN
      L     3;	// Position StHN
      L     #Par.OutPosTarget;
      ==I;
      R     #StCtoHN;
      JC    xxS2;	//--> StHN
// Transition to StLN
      R     #StCtoHN;
      JU    xxS0;	//--> StLN
NETWORK
TITLE = StHN
// Any transition to StHN
xxS2: S     #StHN;
      S     #Par.OutPulseIsOn;
      R     #Par.OutReAdjust;
      L     0;
      T     #Par.OutDelayTime;
      AN    #tmpReport;
      JC    OUT;
      L     B#(4, 2);	//   MessageClass Info "Set HN"
      JU    LOG;
//=== Logic ====
S2:   AN    #Par.OutPulseIsOn;
      JC    S2J1;
      AN    "GCS7_Gr_OutTick200ms";	//Gr.OutTick200ms
      L     #Par.OutDelayTime;
      JC    S2T2;
      +     2;
      T     #Par.OutDelayTime;
S2T2: L     #Par.ParPulseHN;
      >=I;
      =     #tmpTimeEnd;
      R     #Par.OutPulseIsOn;
      R     #Par.tmpOutpLN;
      S     #OutpHold;
      A     #tmpTimeEnd;
      AN    #Par.ParContinuousHN;
      R     #Par.tmpOutpHN;
// Transition to StCtoLN
S2J1: L     #Par.OutPosTarget;
      L     3;	//Position HN; 
      <I;
      R     #StHN;
      JC    xxS3;	//--> StCtoLN
// Transition to StFault
      L     #tmpPosActual;
      ==I;
      A     #tmpPosValid;
      JC    OUT;
      A     #Par.ParNoReAdjust;
      AN    #tmpLocal;
      R     #StHN;
      JC    xxS4;	//-->StFault
// Transition to StCtoHN
      S     #tmpCntReAdjustUp;
      S     #Par.OutReAdjust;
      R     #StHN;
      JU    xxS1;	//-->StCtoHN
NETWORK
TITLE = StCtoLN
// Any transition to StCtoLN
xxS3: S     #StCtoLN;
      S     #Par.tmpOutpLN;
      R     #OutpHold;
      R     #Par.tmpOutpHN;
      AN    #Par.OutPulseIsOn;
      JC    OUT;
      L     0;
      T     #Par.OutDelayTime;
      JU    OUT;
//=== Logic ====
S3:   AN    "GCS7_Gr_OutTick200ms";	//Gr.OutTick200ms
      L     #Par.OutDelayTime;
      JC    S3T2;
      +     2;
      T     #Par.OutDelayTime;
S3T2: L     #Par.ParTransTime;
      >=I;
      O;
      A     #tmpLocal;	//[5.0]
      A     #tmpAnalog;	//[6.0]//[5.0]
      =     #tmpTimeEnd;
// Transition to StNoPos
//      U     #tmpTimeEnd  //[5.2]
      AN    #tmpInpLN;	//[4.1]
      AN    #Par.ParNoLSLN;
      AN    #tmpPosValid;	//[5.0]
      A     #tmpLocal;
      R     #StCtoLN;
      JC    xxS5;	//--> StNoPosition
//Transition A to StLN    
      L     #Par.OutPosTarget;	//                
      L     0;	//Target=StLN
      ==I;
      A     #tmpTimeEnd;
      A(;
      A     #tmpInpLN;	//[4.1]
      O     #Par.ParNoLSLN;
      );
S3S0: R     #StCtoLN;
      JC    xxS0;	//-->StLN
//[4.0 -->
      L     1;	// Target position =StMiddle1
      L     #Par.OutPosTarget;
      <>I;
      A(;
      L     2;	// Target position =StMiddle2
      L     #Par.OutPosTarget;
      <>I;
      );
      ON    #tmpAnalog;	//[6.0]
      O     #tmpLocal;	//[5.0]
      O     #Par.ParAngle;	//[5.0]
//<--4.0]
      A(;
      L     #Par.OutPosTarget;
      L     #tmpPosActual;
      ==I;
      );
      A     #tmpPosValid;
      JC    S3xx;
//Transition to StCtoHN   
      >I;
      A     #tmpPosValid;
      O;
      A     #tmpTimeEnd;
      AN    #Par.OutReAdjust;
      O(;	//[4.0]
      L     #OutPosition;	//[4.0]
      L     #Par.ParPositionTolerance;	//[4.0]
      +I;	//[4.0]
      L     #InPositionMiddle;	//[4.0]
      <I;	//[4.0]
      A(;
      L     1;	// Target position =StMiddle1
      L     #Par.OutPosTarget;
      ==I;
      );
      A     #tmpAnalog;	//[6.0]//[4.0]
      );	//[4.0]
      JC    S3S1;	//-->StCtoHN
//Transition to StFault   
      A     #tmpTimeEnd;
      R     #StCtoLN;
      JC    xxS4;	//-->StFault
      JU    OUT;
// Transition to StMiddle1
S3xx: L     1;	// Target position =StMiddle1
      L     #Par.OutPosTarget;
      ==I;
      R     #StCtoLN;
      JC    xxS6;	//-->StMiddle1
// Transition to StMiddle2
      L     2;	// Target position =StMiddle2
      ==I;
      R     #StCtoLN;
      JC    xxS7;	//-->StMiddle2
// Transition to StHN
      L     3;	// Target position =StHN
      L     #Par.OutPosTarget;
      ==I;
      R     #StCtoLN;
      JC    xxS2;	//-->StHN
// Transition B to StLN
      JU    S3S0;	//-->StLN
// Transition B to StCtoHN
S3S1: A     #Par.OutReAdjust;
      JC    S3x1;
      L     0;
      T     #Par.OutDelayTime;
S3x1: S     #Par.OutReAdjust;
      R     #StCtoLN;
      JU    xxS1;	//-->StCtoHN
NETWORK
TITLE = StFault
// Any transiton to Fault  
xxS4: S     "GCS7_Gr_InFaultFlag";	// Gr.InFaultFlag
      S     #StFault;
      R     #Par.tmpOutpLN;
      R     #OutpHold;
      R     #Par.tmpOutpHN;
      A     #Par.ParNoLSLN;
      R     #Par.OutReAdjust;
      CALL  "SYS_Horn_Code" (
           FcCode                   := 1,
           ParObjectType            := 1020,
           ParObjectNo              := #Par.ParObjectNo,
           ParHornCode              := #Par.ParHornCode);
      L     #Par.OutPosTarget;
      L     B#(1, 11);	//   MessageClass "Fault xxx" (Code=B#(1,11),B#(1,12),B#(1,13),B#(1,14)
      +I;
      AN    #InpFaultAI;
      JC    LOG;
      L     B#(1, 15);	//   MessageClass "Fault Analog Input"
      JU    LOG;
//=== Logic ====
S4:   AN    #tmpLocalFault;
      AN    #CmdFaultReset;
      AN    "GCS7_Gr_OutFaultReset";	// OutFaultReset
      JC    OUT;
      R     #StFault;	//        
      S     #StNoPosition;	//--> StNoPosition
      L     B#(3, 9);	// MessageClass Oper "Fault cancelled" 
      JU    LOG;
NETWORK
TITLE = StNoPosition
// Any transition to StNoPosition
xxS5: S     #StNoPosition;
      R     #Par.tmpOutpLN;
      R     #Par.tmpOutpHN;
      A     #Par.ParNoLSLN;
      R     #Par.OutReAdjust;
      AN    #tmpReport;
      JC    OUT;
      L     B#(4, 5);	//   MessageClass Info "Set no position"
      JU    LOG;
//==Logic==== 
//--Transiton to StCtoLN 
S5:   L     0;
      T     #Par.OutDelayTime;
      A     #tmpNext;
      O     #InLN;	//[5.1]
      AN    #InManual;
      AN    #InLocal;
      O;
      A     #InManual;
      A     #CmdLNMan;
      O     #tmpPosValid;
      R     #StNoPosition;
      JC    xxS3;	//-->StCtoLN
//--Transiton to StCtoHN 
      A     #InManual;
      A     #CmdNextPos;
      R     #StNoPosition;
      JC    xxS1;	//-->StCtoHN
      JU    OUT;
NETWORK
TITLE = StMiddle1 / StMiddle 2
// Any transition to StMiddle1
xxS6: S     #StMiddle1;
      S     #Par.OutPulseIsOn;
      R     #Par.OutReAdjust;
      L     0;
      T     #Par.OutDelayTime;
      AN    #tmpReport;
      JC    OUT;
      L     B#(4, 3);	//   MessageClass Info "SET_Middle1"
      JU    LOG;
// Any transition to StMiddle2
xxS7: S     #StMiddle2;
      S     #Par.OutPulseIsOn;
      R     #Par.OutReAdjust;
      L     0;
      T     #Par.OutDelayTime;
      AN    #tmpReport;
      JC    OUT;
      L     B#(4, 4);	//   MessageClass Info "SET Middle 2"
      JU    LOG;
//==Logic==== 
S7:   L     2;	//Actual state is StMiddle2
      JU    S6S7;
S6:   L     1;	//Actual state is StMiddle1
S6S7: T     #tmpStateNr;
// This part is used for StMiddle1 and StMiddle2
      AN    #Par.OutPulseIsOn;
      JC    S6J1;
      AN    "GCS7_Gr_OutTick200ms";	//Gr.OutTick200ms
      L     #Par.OutDelayTime;
      JC    S6T1;
      +     2;
      T     #Par.OutDelayTime;
S6T1: L     #Par.ParPulseMiddle;
      >=I;
      =     #tmpTimeEnd;
      R     #Par.OutPulseIsOn;
      R     #Par.tmpOutpLN;
      S     #OutpHold;
      R     #Par.tmpOutpHN;
// Transition to StCtoLN
S6J1: L     #Par.OutPosTarget;
      L     #tmpStateNr;
      <I;
S6S3: R     #StMiddle1;
      R     #StMiddle2;
      JC    xxS3;	//--> StCtoLN
// Transition A to StCtoHN
      >I;
S6S1: R     #StMiddle1;
      R     #StMiddle2;
      JC    xxS1;	//--> StCtoHN
// Transition to StFault
      L     #tmpPosActual;
      ==I;
      A     #tmpPosValid;
      JC    OUT;
      A     #Par.ParNoReAdjust;
      AN    #tmpLocal;
      R     #StMiddle1;
      R     #StMiddle2;
      JC    xxS4;	//-->StFault
// Transition B to StCtoLN
      S     #tmpCntReAdjustUp;
      L     #InPositionMiddle;	//[5.0]
      L     #Par.tmpInPosition;	//[5.0]
      >I;	//[5.0]
      A     #tmpAnalog;	//[6.0]
      JC    S6S1;	//--> StCtoHN [5.0]
      JU    S6S3;	//--> StCtoLN
NETWORK
TITLE = Log
LOG:  A     #Par.ParLogOff;	//---Set LOG Message
      JC    OUT;
      T     #tmpLOGvalue;
      L     W#16#FF;
      AW;
      T     #OutAlarmNrLog;
      CALL  "GCS7_LogConvert" (
           ObjectNo                 := #Par.ParObjectNo,
           MsgType                  := #Par.ParMsgType,
           ClassMsgTxt              := #tmpLOGvalue,
           OType                    := 1020);	// LOG Message Converter / Entry / Contains Class and TextNo
NETWORK
TITLE = Global End
// ==Init Outputs
OUT:  A     #tmpLocal;
      R     #OutpHold;
      R     #Par.tmpOutpLN;
      R     #Par.tmpOutpHN;
//=== Output =============
      L     1;	//[3.0]
      L     #Par.OutPosTarget;	//[3.0]
      ==I;	//[3.0]
      O(;	//[3.0]
      L     2;	//[3.0]
      ==I;	//[3.0]
      );	//[3.0]
      =     #tmpMid;	//[3.0]
      AN    #tmpMid;	//[3.0]
      ON    #Par.ParDFZK;	//[3.0]
      A     #Par.tmpOutpLN;	//[3.0]
      =     #OutpLN;	//[3.0]
      A     #tmpMid;	//[3.0]
      A     #Par.tmpOutpHN;	//[3.0]
      O     #Par.tmpOutpLN;	//[3.0]
      A     #Par.ParDFZK;	//[3.0]
      =     #OutpLN2;	//[3.0]
      A     #tmpMid;	//[3.0]
      A     #Par.tmpOutpLN;	//[3.0]
      O     #Par.tmpOutpHN;	//[3.0]
      A     #Par.ParDFZK;	//[3.0]
      =     #OutpHN2;	//[3.0]
      AN    #tmpMid;	//[3.0]
      ON    #Par.ParDFZK;	//[3.0]
      A     #Par.tmpOutpHN;	//[3.0]
      =     #OutpHN;	//[3.0]
//=== Warning =====               
      L     #Par.tmpInPosition;
      L     #InPositionMiddle;
      ==I;
      JC    o3;
      T     #Par.tmpInPosition;
      R     #OutWarning;
      L     0;
      T     #Par.OutCntReAdjust;
o3:   AN    #tmpCntReAdjustUp;
      JC    o4;
      L     #Par.OutCntReAdjust;
      +     1;
      T     #Par.OutCntReAdjust;
o4:   L     #Par.OutWarningTime;
      L     #Par.ParWarningTime;
      <I;
      JC    o5;
      L     0;
      T     #Par.OutCntReAdjust;
      T     #Par.OutWarningTime;
o5:   L     #Par.OutCntReAdjust;
      L     0;
      ==I;
      ON    "GCS7_Gr_OutTick200ms";	//Gr.OutTick200ms
      JC    o6;
      L     #Par.OutWarningTime;
      +     2;
      T     #Par.OutWarningTime;
o6:   L     #Par.OutCntReAdjust;
      L     5;
      >=I;
      S     #OutWarning;
      A     #tmpLocal;
      O     #CmdFaultReset;
      O     "GCS7_Gr_OutFaultReset";	// OutFaultReset [5.3]
      R     #OutWarning;
//=====Clear all commands
      SET;
      R     #CmdLNMan;
      R     #CmdPrevPos;
      R     #CmdNextPos;
      R     #CmdMiddle2;
      R     #CmdMiddle1;
      R     #CmdHN;
      R     #CmdFaultReset;
//--Output for group 
      A     #InDPFault;
      AN    #tmpLocalFault;
      S     "GCS7_Gr_InDPFault";
      A     #InHWStop;
      AN    #tmpLocalFault;
      S     "GCS7_Gr_InHWStop";
NETWORK
TITLE = State Code
      L     1;
      A     #StLN;
      JC    STC1;
      L     2;
      A     #StCtoHN;
      JC    STC1;
      L     3;
      A     #StHN;
      JC    STC1;
      L     4;
      A     #StCtoLN;
      JC    STC1;
      AN    #StNoPosition;
      JC    STCM;
      L     45;	//Code: StNoPosition.HWStop
      A     #InHWStop;
      JC    STC;
      L     55;	//Code: StNoPosition.DPFault
      A     #InDPFault;
      JC    STC;
      L     5;
      JU    STC1;
STCM: L     6;
      A     #StMiddle1;
      JC    STC1;
      L     7;
      A     #StMiddle2;
      JC    STC1;
      L     32;	// Code: fault
      JU    STC;
STC1: AN    #OutWarning;
      JC    STC;
      +     20;
STC:  L     #StCode;	// Old state code
      TAK;
      T     #StCode;	// Save state code
      <>I;
      L     3;	// Load code for CBit methode
      CC    "SYS_CBitCtrl";
END_FUNCTION_BLOCK

FUNCTION_BLOCK "GCS7_E_DMDS"	// FB 21
TITLE = DMDS
//  
//COPYRIGHT:    (C) 1996 BY  BUHLER LTD.
//                           CH-9240 UZWIL  SWITZERLAND
//
//PRODUCT:      GCS7
//
//TITLE:        Element Control DMDS
//
//-------------------------------------------------------------------------
//
//IDENT:        AUTHOR:             DEPT:                       DATE:
//
//FB21.4.1      A. Egli             CT3                         16-Jun-2003
//              Store text number, when calling FC4 
//FB21.4.0      A. Egli             CT3                         17-Jun-2002
//              New Release with one block 
//FB21.2C       A. Egli             CT3                         03-Jun-1999
//              Manual Mode
//FB21.2B       A. Egli             CT3                         25-Mai-1999
//              Gloabl fault reset
//FB21.2A       A. Egli             CT3                         04-Mai-1998
//              StFault = StCode 32
//FB21.1A       A.Egli              AEE61                       28-Jul-1997
//              1st Release in S7
//
//-------------------------------------------------------------------------
//
//PURPOSE:      MANUAL : see [DMDxxMAN]
//
//RESTRICTIONS: S7
//              ACCU2: Pointer to dynamic datas of the element
//              ACCU1: Pointer to parameter datas of the element
//
//-------------------------------------------------------------------------
//
//=======================================================
//Log Message: 
//------------------------------------------------------
//0   closed
//1   fine dosing
//2   full open
//3   coarse dosing
//9   fault cancelled
//10  fault not closed
//11  fault not open
//
//=======================================================
//StCode:  State               
//------------------------------------------------------
//32  StFault               
// 1  StClosed              
//41  StClosed.HWStop               StClosed + InHWStop
//51  StClosed.DPFault              StClosed + InDPFault
// 2  StOpening             
// 3  StCoarse              
// 4  StClosing             
//10  StFine                
//11  StOpen                
//
AUTHOR : EA
FAMILY : GCS7LL
NAME : DMDS
VERSION : 4.1
VAR
  StCode : INT ;	//Element state code
  InEnable : BOOL ;	//Interlocking: 1=Enable to open /0=Intermediate closing
  CmdOpen : BOOL ;	//Command for opening (automatic mode) first fine then coarse
  CmdClose : BOOL ;	//Commamd for closing (automatic mode) first full open then closing
  InFine : BOOL ;	//Fine dosing, don't change from fine to coarse
  spare0004 : BOOL ;
  spare0005 : BOOL ;
  spare0006 : BOOL ;
  InpActive : BOOL ;	//DMDS is active
  CmdCloseMan : BOOL ;	//Pulse to close  (manual mode)
  CmdPrevPos : BOOL ;	//Pulse move to next lower  position in manual mode
  CmdNextPos : BOOL ;	//Pulse move to next higher position in manual mode
  CmdFaultReset : BOOL ;	//Command to reset fault
  InLocal : BOOL ;	//1= Local mode (no fault by start with service switch)
  InManual : BOOL ;	//1= Manual/ 0= Automatic
  InReport : BOOL ;	//Report of all state transitions
  spare0207 : BOOL ;
  InHWStop : BOOL ;	//HW stop is detected, no fault
  InDPFault : BOOL ;	//DP-Fault is detected, no fault
  OutTargetPosOpen : BOOL ;	//Internal flag
  InOutManCoarse : BOOL ;	//Manual mode target position is StCoarse
  spare0404 : BOOL ;
  OutpFine : BOOL ;	//Fine dosing requested
  OutpCoarse : BOOL ;	//Coarse dosing requested
  OutpOpen : BOOL ;	//Full open requested
  StClosed : BOOL ;	//Element is closed
  StOpening : BOOL ;	//Element is opening
  StCoarse : BOOL ;	//Element is coarse dosing
  StClosing : BOOL ;	//Element is closing
  StFault : BOOL ;	//Element has a fault
  StFine : BOOL ;	//Element is fine
  StOpen : BOOL ;	//Element is toggling between 'full open' and 'fine dosing'
  OutAlarmNrLog : INT ;	//Last textnumber send to log
  Par : STRUCT
   ParObjectNo : INT ;	//Is used for communication with PC, e.g. for message
   ParMsgType : INT ;	//Is used for message (translation of state)
   ParHornCode : INT ;	//Is used by horn module
   ParLogOff : BOOL ;	//Report is off
   ParManual : BOOL ;	//Manual mode without interlocking
   ParTransTime : INT ;	//Opening and closing time [1/10s] (StOpening/StClosing)
   ParFineToCoarseTime : INT ;	//After this time element changes from StFine to StCoarse [1/10s]
   ParMonTime : INT ;	//Monitoring time until element change to StFault
   ParCntOpenPulse : INT ;	//Number of pulse open in StOpen
   ParPulseFineTime : INT ;	//Pulse length 'fine'      [1/10s]
   ParPulseOpenTime : INT ;	//Pulse length 'full open' [1/10s]
   OutMonTime : INT ;	//Actual monitoring time
   OutDelayTime : INT ;	//Actual time starting, Closing,fine to coarse, pulse time
   OutCntOpenPulse : INT ;	//Actual counter
  END_STRUCT ;
END_VAR
VAR_TEMP
  tmpLOGvalue : WORD ;	//LOG value
  tmpReport : BOOL ;	//Global LOG all
  tmpOpen : BOOL ;
  tmpOff : BOOL ;
  tmpLenDyn : DINT ;
  tmpFlag : BOOL ;
  tmpTimeEnd : BOOL ;
  tmpMonTime : BOOL ;
  tmpCounter : BYTE ;
  tmpFine : BOOL ;
  tmpLocal : BOOL ;
  tmpFullOpen : BOOL ;
  tmpLocalFault : BOOL ;
END_VAR
BEGIN
NETWORK
TITLE =  Start Global
      L     34;
      T     #tmpLenDyn;	//--> Len dynamic data in byte
NETWORK
TITLE = PC Control
//=== Test Object number =====================
      L     "SYS_DirectCtrlDB".PC.ObjectNo;	//PCControl.ObjectNo
      L     #Par.ParObjectNo;	//Input ObjectNo
      <>I;
      JC    Ctrl;
//=== Test OType      ========================
      L     1021;	//Input object type
      L     "SYS_DirectCtrlDB".PC.ObjectType;	//PCControl.ObjectType
      <>I;
      JC    Ctrl;
//=== Test Handshake =========================
      A     "SYS_DirectCtrlDB".PC.Hsk.FExamine;	// Handshake.FExamine
      JC    pExa;
      A     "SYS_DirectCtrlDB".PC.Hsk.FDefineCmd;	// Handshake.FDefineCmd
      JC    pCmd;
      A     "SYS_DirectCtrlDB".PC.Hsk.FDefinePara;	// Handshake.FDefinePara
      JC    pPar;
pIni: L     2;	// FcInit
      UC    "SYS_DirectCtrl";
      JU    Ctrl;
// Write parameter 
pPar: LAR1  P#DBX 58.0;	//PCControl.Value[1]
      L     P##Par;
      L     DW#16#FFFFF;
      AD;
      +AR1;
      L     DBW [AR1,P#8.0];
      T     #Par.ParTransTime;
      L     DBW [AR1,P#10.0];
      T     #Par.ParFineToCoarseTime;
      L     DBW [AR1,P#12.0];
      T     #Par.ParMonTime;
      L     DBW [AR1,P#14.0];
      T     #Par.ParCntOpenPulse;
      L     DBW [AR1,P#16.0];
      T     #Par.ParPulseFineTime;
      L     DBW [AR1,P#18.0];
      T     #Par.ParPulseOpenTime;
// Write new commands from PC to Interface of group 
pCmd: A     "SYS_DirectCtrlDB".PC.Cmd1[1];	//Cmd1[1]   =CmdOpen
      S     #CmdOpen;
      A     "SYS_DirectCtrlDB".PC.Cmd1[2];	//Cmd1[2]   =CmdClose  
      S     #CmdClose;
      A     "SYS_DirectCtrlDB".PC.Cmd1[8];	//Cmd1[8]   =CmdCloseMan
      S     #CmdCloseMan;
      A     "SYS_DirectCtrlDB".PC.Cmd1[9];	//Cmd1[9]   =CmdNextPos
      S     #CmdPrevPos;
      A     "SYS_DirectCtrlDB".PC.Cmd1[10];	//Cmd1[10]   =CmdPrevPos
      S     #CmdNextPos;
      A     "SYS_DirectCtrlDB".PC.Cmd1[11];	//Cmd1[11] =CmdFaultReset
      S     #CmdFaultReset;
      A     "SYS_DirectCtrlDB".PC.Cmd1[13];	//Cmd1[13] =CmdManualOn
      S     #InManual;
      A     "SYS_DirectCtrlDB".PC.Cmd2[13];	//Cmd2[13] =CmdManualOff
      R     #InManual;
      A     "SYS_DirectCtrlDB".PC.Cmd1[14];	//Cmd1[14]=CmdReportOn
      S     #InReport;
      A     "SYS_DirectCtrlDB".PC.Cmd2[14];	//Cmd2[14]=CmdReportOff
      R     #InReport;
      JU    pIni;
pExa: TAR2;	// Address Dynamic datas
      T     "SYS_DirectCtrlDB".GC.InDynAddr;	// -->PCControl.GC.InDynAddr
      L     #tmpLenDyn;	// Length Dynamic datas
      T     "SYS_DirectCtrlDB".GC.InDynLen;	// -->PCControl.GC.InDynLen
      L     0;
      T     "SYS_DirectCtrlDB".GC.InParaAddr;	// -->PCControl.GC.InParaAddr
      T     "SYS_DirectCtrlDB".GC.InParaLen;	// -->PCControl.GC.InParaLen
      L     1;	// Code FcExamine
      UC    "SYS_DirectCtrl";
      L     10;	//Revision
      T     "SYS_DirectCtrlDB".GC.Revision;
NETWORK
TITLE =  All State Init
//===Clear tmp Variable
//===Global Group Orders===
Ctrl: A     "GCS7_Gr_OutManualOn";	//Gr.OutManualOn
      S     #InManual;
      A     "GCS7_Gr_OutManualOff";	//Gr.OutManualOff
      R     #InManual;
      A     #InManual;
      S     "GCS7_Gr_InManual";	//Gr.InManualMode
//---Report is on---
      A     "GCS7_Gr_OutReportAll";	//Gr.OutReportAll
      O     #InReport;
      =     #tmpReport;
      A     #InLocal;
      AN    #InManual;
      =     #tmpLocalFault;
      A     #tmpLocalFault;
      O     #InHWStop;
      O     #InDPFault;
      =     #tmpLocal;
//---Enable---
      AN    #InEnable;
      AN    #InManual;
      O;
      AN    #InEnable;
      AN    #Par.ParManual;
      A     #InManual;
      O;
      A     #StFine;
      A     #CmdPrevPos;
      A     #InManual;
      O     #tmpLocal;
      O     #CmdCloseMan;
      =     #tmpOff;
//Full Open
      AN    #InManual;
      A     #CmdClose;
      O;
      A     #InManual;
      A     #StCoarse;
      A     #CmdNextPos;
      =     #tmpFullOpen;
//---Fine/Coarse---
      A     #StFine;
      A     #CmdNextPos;
      S     #InOutManCoarse;
      A     #StCoarse;
      A     #CmdPrevPos;
      O     #StClosed;
      O     #StFault;
      ON    #InManual;
      O     #tmpOff;
      R     #InOutManCoarse;
      A     #InFine;
      AN    #InManual;
      O;
      AN    #InOutManCoarse;
      A     #InManual;
      =     #tmpFine;
//---Opening---
      A(;
      A     #CmdOpen;
      AN    #InManual;
      O     #CmdNextPos;
      O;
      A     #StOpen;
      A     #CmdPrevPos;
      );
      AN    #tmpOff;
      =     #tmpOpen;
//--- Init in local mode  
      A     #tmpLocal;
      O     #tmpOff;
      R     #OutpFine;
      R     #OutpCoarse;
      R     #OutpOpen;
NETWORK
TITLE = States
//===State machine===
      A     #StClosed;
      JC    S0;
      A     #StOpening;
      JC    S1;
      A     #StCoarse;
      JC    S2;
      A     #StClosing;
      JC    S3;
      A     #StFault;
      JC    S4;
      A     #StFine;
      JC    S5;
      A     #StOpen;
      JC    S6;
      S     #StClosed;	// Init
      L     0;
      T     #Par.OutMonTime;
      JU    S0;
NETWORK
TITLE = StClosed
// Any transition to StClosed
xxS0: S     #StClosed;
      L     0;
      T     #Par.OutMonTime;
      AN    #tmpReport;
      JC    OUT;
      L     B#(4, 0);	// MessageClass Info "closed" 
      JU    LOG;
//=== Logic ====
S0:   L     #Par.ParMonTime;
      L     #Par.OutMonTime;
      <=I;
      A     #InpActive;
      AN    #tmpLocal;
      =     #tmpMonTime;	//Condition for fault
      AN    #InpActive;
      O     #tmpLocal;
      ON    "GCS7_Gr_OutTick200ms";	//Gr.OutTick200ms
      JC    S0N1;
      L     #Par.OutMonTime;
      +     2;
      T     #Par.OutMonTime;
S0N1: A     #InpActive;
      JC    S0N2;
      L     0;
      T     #Par.OutMonTime;
// Transition to StOpening (active) 
S0N2: A     #tmpOpen;
      AN    #tmpLocal;
      R     #StClosed;
      JC    xxS1;	//--> StOpening
// Transition to StOpening (local) 
      A     #InpActive;
      A     #tmpLocal;
      R     #StClosed;
      JC    xxS1;
// Transition to fault
      AN    #tmpMonTime;
      JC    OUT;
      R     #StClosed;
      L     B#(1, 10);	// Message ('Fault not closed' )
      JU    xxS4;
NETWORK
TITLE = StOpening
// Any transition to StOpening
xxS1: S     #StOpening;
      R     #OutpCoarse;
      L     0;
      T     #Par.OutDelayTime;
      A     #tmpOpen;
      R     #OutTargetPosOpen;
      =     #OutpFine;
      A     #tmpFullOpen;
      S     #OutTargetPosOpen;
      =     #OutpOpen;
      R     #OutpFine;
      JU    OUT;
//=== Logic ====
S1:   AN    "GCS7_Gr_OutTick200ms";	//Gr.OutTick200ms
      L     #Par.OutDelayTime;
      JC    S1_1;
      +     2;
      T     #Par.OutDelayTime;
S1_1: L     #Par.ParTransTime;
      >=I;
      =     #tmpFlag;	// End transition time
// Transition for StClosing
      AN    #InpActive;
      A     #tmpLocal;
      O;
      A     #tmpOff;
      AN    #tmpLocal;
      R     #StOpening;
      JC    xxS3;	//--> StClosing 
// Transition for StFine
      AN    #OutTargetPosOpen;
      O     #tmpLocal;
      A     #tmpFlag;
      A     #InpActive;
      R     #StOpening;
      JC    xxS5;	//--> StFine
// Transition for StOpen
      A     #tmpFlag;
      A     #InpActive;
      R     #StOpening;
      JC    xxS6;	//--> StFullOpen
// Transition for StFault
      O     #InpActive;
      ON    #tmpFlag;
      JC    OUT;
// Transition to StFault
      R     #StOpening;
      S     #StFault;
      L     0;
      T     #Par.OutDelayTime;
      T     #Par.OutMonTime;
      L     B#(1, 11);	// Message ('Fault not open' )
      JU    xxS4;
NETWORK
TITLE = StCoarse
// Any transition to StCoarse
xxS2: S     #StCoarse;
      R     #OutpFine;
      R     #OutpCoarse;
      R     #OutpOpen;
      L     0;
      T     #Par.OutMonTime;
      AN    #tmpLocal;
      S     #OutpCoarse;
      AN    #tmpReport;
      JC    OUT;
      L     B#(1, 3);	// Message ('Started coarse' )
      JU    LOG;
//=== Logic ====
S2:   L     #Par.ParMonTime;
      L     #Par.OutMonTime;
      <=I;
      AN    #InpActive;
      AN    #tmpLocal;
      =     #tmpMonTime;	// Transition for fault
      A     #InpActive;
      O     #tmpLocal;
      ON    "GCS7_Gr_OutTick200ms";	//Gr.OutTick200ms
      JC    S2A1;
      L     #Par.OutMonTime;
      +     2;
      T     #Par.OutMonTime;
S2A1: AN    #InpActive;
      JC    S2A2;
      L     0;
      T     #Par.OutMonTime;
// Transition to StOpen
S2A2: A     #tmpFullOpen;
      AN    #tmpLocal;
      R     #StCoarse;
      JC    xxS6;	//--> StFullOpen
      A     #tmpFine;
      R     #StCoarse;
      JC    xxS5;	//--> StFine
// Transition to StClosing
      AN    #InpActive;
      A     #tmpLocal;
      O;
      A     #tmpOff;
      AN    #tmpLocal;
      R     #StCoarse;
      JC    xxS3;	//--> StClosing
// Transition for fault
      AN    #tmpMonTime;
      JC    OUT;
      R     #StCoarse;
      L     B#(1, 11);	// Message ('Fault not open' )
      JU    xxS4;
NETWORK
TITLE = StClosing
// Any Transition to StClosing
xxS3: S     #StClosing;
      R     #OutpFine;
      R     #OutpCoarse;
      R     #OutpOpen;
      L     0;
      T     #Par.OutDelayTime;
      JU    OUT;
//=== Logic ====
S3:   AN    "GCS7_Gr_OutTick200ms";	//Gr.OutTick200ms
      L     #Par.OutDelayTime;
      JC    S31T;
      +     2;
      T     #Par.OutDelayTime;
S31T: L     #Par.ParTransTime;
      >=I;
      =     #tmpFlag;
// Transition for StClosed
      A     #tmpFlag;
      AN    #InpActive;
      R     #StClosing;
      JC    xxS0;
// Transition for StOpening
      A     #tmpLocal;
      A     #InpActive;
      A     #tmpFlag;
      O     #tmpOpen;
      R     #StClosing;
      JC    xxS1;
// Transition for StFault
      AN    #tmpFlag;
      JC    OUT;
      R     #StClosing;
      L     B#(1, 10);	// Message ('Fault not closed' )
      JU    xxS4;
NETWORK
TITLE = StFault
// Any transiton to Fault  
xxS4: S     "GCS7_Gr_InFaultFlag";	// Gr.InFaultFlag
      S     #StFault;
      R     #OutpFine;
      R     #OutpCoarse;
      R     #OutpOpen;
      S     #StFault;
      T     #tmpLOGvalue;	//[4.1]
      CALL  "SYS_Horn_Code" (
           FcCode                   := 1,
           ParObjectType            := 1021,
           ParObjectNo              := #Par.ParObjectNo,
           ParHornCode              := #Par.ParHornCode);
      L     #tmpLOGvalue;	//[4.1]
      JU    LOG;
//=== Logic ====
S4:   AN    #CmdFaultReset;
      AN    "GCS7_Gr_OutFaultReset";	// OutFaultReset
      AN    #tmpLocalFault;
      JC    OUT;
// retry of fault message
      A     #InpActive;
      AN    #tmpLocal;
      L     B#(1, 10);	// Message ('fault not closed' )
      JC    LOG;
//Transition to StClosed
      R     #StFault;
      S     #StClosed;
      L     0;
      T     #Par.OutMonTime;
      L     B#(3, 9);	// Message ('fault cancelled' )
      JU    LOG;
NETWORK
TITLE = StFine
// Any transition to StFine
xxS5: S     #StFine;
      R     #OutpCoarse;
      R     #OutpOpen;
      AN    #tmpLocal;
      =     #OutpFine;
      L     0;
      T     #Par.OutDelayTime;
      T     #Par.OutMonTime;
      AN    #tmpReport;
      JC    OUT;
      L     B#(4, 1);	// MessageClass Info "Started fine" 
      JU    LOG;
//=== Logic ====
S5:   AN    "GCS7_Gr_OutTick200ms";	//Gr.OutTick200ms
      O     #tmpFine;
      L     #Par.OutDelayTime;
      JC    S55T;
      +     2;
      T     #Par.OutDelayTime;
S55T: L     #Par.ParFineToCoarseTime;
      >=I;
      =     #tmpTimeEnd;
      L     #Par.ParMonTime;
      L     #Par.OutMonTime;
      <=I;
      AN    #InpActive;
      AN    #tmpLocal;
      =     #tmpFlag;	// Transition for fault
      A     #InpActive;
      O     #tmpLocal;
      ON    "GCS7_Gr_OutTick200ms";	//Gr.OutTick200ms
      JC    S5_1;
      L     #Par.OutMonTime;
      +     2;
      T     #Par.OutMonTime;
S5_1: AN    #InpActive;
      JC    S5_2;
      L     0;
      T     #Par.OutMonTime;
// Transition for StClosing
S5_2: AN    #InpActive;
      A     #tmpLocal;
      O;
      A     #tmpOff;
      AN    #tmpLocal;
      R     #StFine;
      JC    xxS3;	//--> StClosing
// Transition for StOpen
      A     #tmpFullOpen;
      AN    #tmpOpen;
      AN    #tmpLocal;
      R     #StFine;
      JC    xxS6;	//--> StFullOpen
// Transition for StCoarse
      A     #tmpTimeEnd;
      AN    #tmpFine;
      R     #StFine;
      JC    xxS2;	// Transition to StCoarse
// Transition for StFault 
      AN    #tmpFlag;
      O     #tmpLocal;
      JC    OUT;
      R     #StFine;
      L     B#(1, 11);	// Message ('fault not open' )
      JU    xxS4;
NETWORK
TITLE = StOpen
// Any transition to StOpen
xxS6: S     #StOpen;
      R     #OutpFine;
      R     #OutpCoarse;
      S     #OutpOpen;
      L     0;
      T     #Par.OutMonTime;
      T     #Par.OutCntOpenPulse;
      T     #Par.OutDelayTime;
      AN    #tmpReport;
      JC    OUT;
      L     B#(4, 2);	// MessageClass Info "Full open" 
      JU    LOG;
//=== Logic ====
S6:   AN    "GCS7_Gr_OutTick200ms";	//Gr.OutTick200ms
      L     #Par.OutDelayTime;
      JC    S6T2;
      +     2;
      T     #Par.OutDelayTime;
S6T2: L     #Par.ParPulseOpenTime;
      <I;	// Pulse time finsehed
      ON    #OutpOpen;
      JC    S6T3;
      R     #OutpCoarse;
      R     #OutpOpen;
      S     #OutpFine;
      L     0;
      T     #Par.OutDelayTime;
      L     #Par.OutCntOpenPulse;
      +     1;
      T     #Par.OutCntOpenPulse;
      JU    S6T4;
S6T3: L     #Par.OutDelayTime;
      L     #Par.ParPulseFineTime;
      <I;	// Pausing time finished
      O     #OutpOpen;
      JC    S6T4;
      R     #OutpFine;
      R     #OutpCoarse;
      S     #OutpOpen;
      L     0;
      T     #Par.OutDelayTime;
S6T4: L     #Par.ParMonTime;
      L     #Par.OutMonTime;
      <=I;
      AN    #InpActive;
      AN    #tmpLocal;
      =     #tmpFlag;
// Transition for fault
      A     #InpActive;
      O     #tmpLocal;
      ON    "GCS7_Gr_OutTick200ms";	//Gr.OutTick200ms
      JC    S6F1;
      L     #Par.OutMonTime;
      +     2;
      T     #Par.OutMonTime;
S6F1: AN    #InpActive;
      JC    S6F2;
      L     0;
      T     #Par.OutMonTime;
// Transition to StClosing
S6F2: A     #tmpOff;
      O(;
      L     #Par.OutCntOpenPulse;
      L     #Par.ParCntOpenPulse;
      >=I;
      );
      O     #tmpLocal;
// Transition to StClosing
      R     #StOpen;
      JC    xxS3;	//--> StClosing
// Transition for StFine
      A     #tmpOpen;
// Transition to StClosing
      R     #StOpen;
      JC    xxS5;	//--> StFine
// Transition for Fault
      AN    #tmpFlag;
      JC    OUT;
      R     #StOpen;
      L     B#(1, 11);	// Message ('Fault not open' )
      JU    xxS4;	//--> StFault
NETWORK
TITLE = Log
LOG:  A     #Par.ParLogOff;	//---Set LOG Message
      JC    OUT;
      T     #tmpLOGvalue;
      L     W#16#FF;
      AW;
      T     #OutAlarmNrLog;
      CALL  "GCS7_LogConvert" (
           ObjectNo                 := #Par.ParObjectNo,
           MsgType                  := #Par.ParMsgType,
           ClassMsgTxt              := #tmpLOGvalue,
           OType                    := 1021);	// LOG Message Converter / Entry / Contains Class and TextNo
NETWORK
TITLE = Global End
OUT:  SET;	//---Clear all commands
      R     #CmdOpen;
      R     #CmdClose;
      R     #CmdCloseMan;
      R     #CmdPrevPos;
      R     #CmdNextPos;
      R     #CmdFaultReset;
//--Output for group 
      AN    #InLocal;
      O     #InManual;
      A     #InDPFault;
      S     "GCS7_Gr_InDPFault";
      AN    #InLocal;
      O     #InManual;
      A     #InHWStop;
      S     "GCS7_Gr_InHWStop";
NETWORK
TITLE = State Code
      AN    #StClosed;
      JC    STC2;
      L     41;	//Code: StClosed.HWStop
      A     #InHWStop;
      JC    STC;
      L     51;	//Code: StClosed.DPFault
      A     #InDPFault;
      JC    STC;
      L     1;	// Code: closed
      JU    STC;
STC2: L     2;	// Code: opening
      A     #StOpening;
      JC    STC;
      L     3;	// Code: Coarse
      A     #StCoarse;
      JC    STC;
      L     4;	// Code: Closing
      A     #StClosing;
      JC    STC;
      L     10;	// Code: Fine
      A     #StFine;
      JC    STC;
      L     11;	// Code: Full open
      A     #StOpen;
      JC    STC;
      L     32;	// Code: fault
STC:  L     #StCode;	// Old state code
      TAK;
      T     #StCode;	// Save state code
      <>I;
      L     3;	// Load code for CBit methode
      CC    "SYS_CBitCtrl";
END_FUNCTION_BLOCK

